LIN {X 0,Y 475.877,Z 329.982,A -85,B 0,C 180,E1 -7309.364,E2 -7309.364} C_VEL
LIN {X 0,Y 476.76,Z 310.728,A -85,B 0,C 180,E1 -7312.766,E2 -7312.766} C_VEL
LIN {X 0,Y 476.384,Z 304.918,A -85,B 0,C 180,E1 -7313.84,E2 -7313.84} C_VEL
LIN {X 0,Y 474.637,Z 296.366,A -85,B 0,C 180,E1 -7315.548,E2 -7315.548} C_VEL
LIN {X 0,Y 474.643,Z 296.366,A -85,B 0,C 180,E1 -7318.283,E2 -7318.283} C_VEL
LIN {X 0,Y 474.601,Z 296.37,A -85,B 0,C 180,E1 -7321.218,E2 -7321.218} C_VEL
LIN {X 0,Y 474.634,Z 296.366,A -85,B 0,C 180,E1 -7324.241,E2 -7324.241} C_VEL
LIN {X 0,Y 474.587,Z 296.366,A -85,B 0,C 180,E1 -7327.384,E2 -7327.384} C_VEL
LIN {X 0,Y 474.616,Z 296.363,A -85,B 0,C 180,E1 -7330.658,E2 -7330.658} C_VEL
LIN {X 0,Y 474.592,Z 296.363,A -85,B 0,C 180,E1 -7333.48,E2 -7333.48} C_VEL
LIN {X 0,Y 474.593,Z 296.37,A -85,B 0,C 180,E1 -7336.52,E2 -7336.52} C_VEL
LIN {X 0,Y 474.616,Z 296.36,A -85,B 0,C 180,E1 -7339.342,E2 -7339.342} C_VEL
LIN {X 0,Y 474.586,Z 296.37,A -85,B 0,C 180,E1 -7342.616,E2 -7342.616} C_VEL
LIN {X 0,Y 474.632,Z 296.357,A -85,B 0,C 180,E1 -7345.759,E2 -7345.759} C_VEL
LIN {X 0,Y 474.599,Z 296.366,A -85,B 0,C 180,E1 -7348.782,E2 -7348.782} C_VEL
LIN {X 0,Y 474.621,Z 296.358,A -85,B 0,C 180,E1 -7351.716,E2 -7351.716} C_VEL
LIN {X 0,Y 474.629,Z 296.36,A -85,B 0,C 180,E1 -7354.589,E2 -7354.589} C_VEL
LIN {X 0,Y 474.601,Z 296.368,A -85,B 0,C 180,E1 -7357.355,E2 -7357.355} C_VEL
LIN {X 0,Y 474.655,Z 296.355,A -85,B 0,C 180,E1 -7360.09,E2 -7360.09} C_VEL
LIN {X 0,Y 474.639,Z 296.356,A -85,B 0,C 180,E1 -7362.774,E2 -7362.774} C_VEL
LIN {X 0,Y 474.647,Z 296.362,A -85,B 0,C 180,E1 -7365.421,E2 -7365.421} C_VEL
LIN {X 0,Y 474.705,Z 296.35,A -85,B 0,C 180,E1 -7368.038,E2 -7368.038} C_VEL
LIN {X 0,Y 474.711,Z 296.35,A -85,B 0,C 180,E1 -7371.486,E2 -7371.486} C_VEL
LIN {X 0,Y 474.768,Z 296.344,A -85,B 0,C 180,E1 -7374.052,E2 -7374.052} C_VEL
LIN {X 0,Y 474.884,Z 296.325,A -85,B 0,C 180,E1 -7377.455,E2 -7377.455} C_VEL
LIN {X 0,Y 474.911,Z 296.327,A -85,B 0,C 180,E1 -7380,E2 -7380} C_VEL
LIN {X 0,Y 474.885,Z 296.329,A -85,B 0,C 180,E1 -7382.545,E2 -7382.545} C_VEL
LIN {X 0,Y 474.759,Z 296.342,A -85,B 0,C 180,E1 -7385.948,E2 -7385.948} C_VEL
LIN {X 0,Y 474.713,Z 296.351,A -85,B 0,C 180,E1 -7388.514,E2 -7388.514} C_VEL
LIN {X 0,Y 474.706,Z 296.35,A -85,B 0,C 180,E1 -7391.963,E2 -7391.963} C_VEL
LIN {X 0,Y 474.701,Z 296.35,A -85,B 0,C 180,E1 -7395.456,E2 -7395.456} C_VEL
LIN {X 0,Y 474.664,Z 296.36,A -85,B 0,C 180,E1 -7399.011,E2 -7399.011} C_VEL
LIN {X 0,Y 474.59,Z 296.361,A -85,B 0,C 180,E1 -7401.729,E2 -7401.729} C_VEL
LIN {X 0,Y 474.638,Z 296.358,A -85,B 0,C 180,E1 -7404.494,E2 -7404.494} C_VEL
LIN {X 0,Y 474.639,Z 296.361,A -85,B 0,C 180,E1 -7407.324,E2 -7407.324} C_VEL
LIN {X 0,Y 474.604,Z 296.361,A -85,B 0,C 180,E1 -7410.231,E2 -7410.231} C_VEL
LIN {X 0,Y 474.627,Z 296.365,A -85,B 0,C 180,E1 -7413.222,E2 -7413.222} C_VEL
LIN {X 0,Y 474.587,Z 296.364,A -85,B 0,C 180,E1 -7416.324,E2 -7416.324} C_VEL
LIN {X 0,Y 474.629,Z 296.365,A -85,B 0,C 180,E1 -7419.548,E2 -7419.548} C_VEL
LIN {X 0,Y 474.603,Z 296.364,A -85,B 0,C 180,E1 -7422.234,E2 -7422.234} C_VEL
LIN {X 0,Y 474.619,Z 296.363,A -85,B 0,C 180,E1 -7425.298,E2 -7425.298} C_VEL
LIN {X 0,Y 474.607,Z 296.368,A -85,B 0,C 180,E1 -7428.213,E2 -7428.213} C_VEL
LIN {X 0,Y 474.611,Z 296.367,A -85,B 0,C 180,E1 -7431.542,E2 -7431.542} C_VEL
LIN {X 0,Y 474.622,Z 296.365,A -85,B 0,C 180,E1 -7434.725,E2 -7434.725} C_VEL
LIN {X 0,Y 474.664,Z 296.454,A -85,B 0,C 180,E1 -7437.643,E2 -7437.643} C_VEL
LIN {X 0,Y 475.735,Z 302.876,A -85,B 0,C 180,E1 -7438.963,E2 -7438.963} C_VEL
LIN {X 0,Y 475.519,Z 316.144,A -85,B 0,C 180,E1 -7441.533,E2 -7441.533} C_VEL
LIN {X 0,Y 475.428,Z 319.942,A -85,B 0,C 180,E1 -7442.241,E2 -7442.241} C_VEL
LIN {X 0,Y 478.338,Z 335.26,A -85,B 0,C 180,E1 -7442.595,E2 -7442.595} C_VEL
LIN {X 0,Y 477.897,Z 378.829,A -85,B 0,C 180,E1 -7443.253,E2 -7443.253} C_VEL
LIN {X 0,Y 477.216,Z 384.671,A -85,B 0,C 180,E1 -7443.318,E2 -7443.318} C_VEL
LIN {X 0,Y 471.64,Z 403.685,A -85,B 0,C 180,E1 -7443.406,E2 -7443.406} C_VEL
LIN {X 0,Y 470.928,Z 409.529,A -85,B 0,C 180,E1 -7443.471,E2 -7443.471} C_VEL
LIN {X 0,Y 470.678,Z 429.482,A -85,B 0,C 180,E1 -7443.814,E2 -7443.814} C_VEL
LIN {X 0,Y 470.338,Z 442.898,A -85,B 0,C 180,E1 -7444.225,E2 -7444.225} C_VEL
LIN {X 0,Y 469.966,Z 454.955,A -85,B 0,C 180,E1 -7444.773,E2 -7444.773} C_VEL
LIN {X 0,Y 469.553,Z 466.283,A -85,B 0,C 180,E1 -7445.459,E2 -7445.459} C_VEL
LIN {X 0,Y 469.015,Z 478.056,A -85,B 0,C 180,E1 -7446.369,E2 -7446.369} C_VEL
LIN {X 0,Y 468.434,Z 488.504,A -85,B 0,C 180,E1 -7447.39,E2 -7447.39} C_VEL
LIN {X 0,Y 467.969,Z 498.494,A -85,B 0,C 180,E1 -7448.611,E2 -7448.611} C_VEL
LIN {X 0,Y 467.554,Z 506.223,A -85,B 0,C 180,E1 -7449.774,E2 -7449.774} C_VEL
LIN {X 0,Y 467.232,Z 513.348,A -85,B 0,C 180,E1 -7451.096,E2 -7451.096} C_VEL
LIN {X 0,Y 466.966,Z 519.248,A -85,B 0,C 180,E1 -7452.481,E2 -7452.481} C_VEL
LIN {X 0,Y 466.822,Z 523.709,A -85,B 0,C 180,E1 -7453.828,E2 -7453.828} C_VEL
LIN {X 0,Y 466.693,Z 527.025,A -85,B 0,C 180,E1 -7455.166,E2 -7455.166} C_VEL
LIN {X 0,Y 466.599,Z 528.656,A -85,B 0,C 180,E1 -7456.054,E2 -7456.054} C_VEL
LIN {X 0,Y 466.586,Z 529.862,A -85,B 0,C 180,E1 -7456.941,E2 -7456.941} C_VEL
LIN {X 0,Y 466.654,Z 530.818,A -85,B 0,C 180,E1 -7458.219,E2 -7458.219} C_VEL
LIN {X 0,Y 466.597,Z 530.896,A -85,B 0,C 180,E1 -7459.586,E2 -7459.586} C_VEL
LIN {X 0,Y 466.539,Z 530.442,A -85,B 0,C 180,E1 -7460.461,E2 -7460.461} C_VEL
LIN {X 0,Y 466.604,Z 529.545,A -85,B 0,C 180,E1 -7461.337,E2 -7461.337} C_VEL
LIN {X 0,Y 466.652,Z 528.255,A -85,B 0,C 180,E1 -7462.209,E2 -7462.209} C_VEL
LIN {X 0,Y 466.769,Z 525.339,A -85,B 0,C 180,E1 -7463.591,E2 -7463.591} C_VEL
LIN {X 0,Y 466.848,Z 521.789,A -85,B 0,C 180,E1 -7464.817,E2 -7464.817} C_VEL
LIN {X 0,Y 467.051,Z 516.937,A -85,B 0,C 180,E1 -7466.117,E2 -7466.117} C_VEL
LIN {X 0,Y 467.208,Z 510.853,A -85,B 0,C 180,E1 -7467.413,E2 -7467.413} C_VEL
LIN {X 0,Y 467.658,Z 503.274,A -85,B 0,C 180,E1 -7468.708,E2 -7468.708} C_VEL
LIN {X 0,Y 468.057,Z 493.792,A -85,B 0,C 180,E1 -7469.999,E2 -7469.999} C_VEL
LIN {X 0,Y 468.476,Z 484.032,A -85,B 0,C 180,E1 -7471.074,E2 -7471.074} C_VEL
LIN {X 0,Y 469.078,Z 473.058,A -85,B 0,C 180,E1 -7472.039,E2 -7472.039} C_VEL
LIN {X 0,Y 469.529,Z 462.354,A -85,B 0,C 180,E1 -7472.788,E2 -7472.788} C_VEL
LIN {X 0,Y 469.924,Z 449.501,A -85,B 0,C 180,E1 -7473.483,E2 -7473.483} C_VEL
LIN {X 0,Y 470.231,Z 437.091,A -85,B 0,C 180,E1 -7473.963,E2 -7473.963} C_VEL
LIN {X 0,Y 470.484,Z 424.139,A -85,B 0,C 180,E1 -7474.283,E2 -7474.283} C_VEL
LIN {X 0,Y 471.164,Z 335.118,A -85,B 0,C 180,E1 -7475.65,E2 -7475.65} C_VEL
LIN {X 0,Y 468.27,Z 320.023,A -85,B 0,C 180,E1 -7475.996,E2 -7475.996} C_VEL
LIN {X 0,Y 468.872,Z 306.744,A -85,B 0,C 180,E1 -7478.62,E2 -7478.62} C_VEL
LIN {X 0,Y 468.41,Z 301.4,A -85,B 0,C 180,E1 -7479.717,E2 -7479.717} C_VEL
LIN {X 0,Y 467.644,Z 297.234,A -85,B 0,C 180,E1 -7480.608,E2 -7480.608} C_VEL
LIN {X 0,Y 467.588,Z 297.24,A -85,B 0,C 180,E1 -7483.029,E2 -7483.029} C_VEL
LIN {X 0,Y 467.602,Z 297.24,A -85,B 0,C 180,E1 -7485.863,E2 -7485.863} C_VEL
LIN {X 0,Y 467.62,Z 297.231,A -85,B 0,C 180,E1 -7489.307,E2 -7489.307} C_VEL
LIN {X 0,Y 467.535,Z 297.249,A -85,B 0,C 180,E1 -7492.073,E2 -7492.073} C_VEL
LIN {X 0,Y 467.555,Z 297.24,A -85,B 0,C 180,E1 -7494.889,E2 -7494.889} C_VEL
LIN {X 0,Y 467.543,Z 297.242,A -85,B 0,C 180,E1 -7497.773,E2 -7497.773} C_VEL
LIN {X 0,Y 467.542,Z 297.242,A -85,B 0,C 180,E1 -7501.038,E2 -7501.038} C_VEL
LIN {X 0,Y 467.574,Z 297.241,A -85,B 0,C 180,E1 -7504.239,E2 -7504.239} C_VEL
LIN {X 0,Y 467.519,Z 297.245,A -85,B 0,C 180,E1 -7507.181,E2 -7507.181} C_VEL
LIN {X 0,Y 467.552,Z 297.242,A -85,B 0,C 180,E1 -7510.266,E2 -7510.266} C_VEL
LIN {X 0,Y 467.513,Z 297.249,A -85,B 0,C 180,E1 -7512.567,E2 -7512.567} C_VEL
LIN {X 0,Y 467.557,Z 297.245,A -85,B 0,C 180,E1 -7515.051,E2 -7515.051} C_VEL
LIN {X 0,Y 467.555,Z 297.244,A -85,B 0,C 180,E1 -7518.725,E2 -7518.725} C_VEL
LIN {X 0,Y 467.538,Z 297.241,A -85,B 0,C 180,E1 -7521.952,E2 -7521.952} C_VEL
LIN {X 0,Y 467.54,Z 297.249,A -85,B 0,C 180,E1 -7525.165,E2 -7525.165} C_VEL
LIN {X 0,Y 467.535,Z 297.241,A -85,B 0,C 180,E1 -7528.256,E2 -7528.256} C_VEL
LIN {X 0,Y 467.518,Z 297.25,A -85,B 0,C 180,E1 -7531.246,E2 -7531.246} C_VEL
LIN {X 0,Y 467.553,Z 297.239,A -85,B 0,C 180,E1 -7534.405,E2 -7534.405} C_VEL
LIN {X 0,Y 467.563,Z 297.239,A -85,B 0,C 180,E1 -7536.995,E2 -7536.995} C_VEL
LIN {X 0,Y 467.608,Z 297.24,A -85,B 0,C 180,E1 -7539.776,E2 -7539.776} C_VEL
LIN {X 0,Y 467.546,Z 297.241,A -85,B 0,C 180,E1 -7542.504,E2 -7542.504} C_VEL
LIN {X 0,Y 467.55,Z 297.24,A -85,B 0,C 180,E1 -7545.194,E2 -7545.194} C_VEL
LIN {X 0,Y 467.638,Z 297.236,A -85,B 0,C 180,E1 -7547.854,E2 -7547.854} C_VEL
LIN {X 0,Y 467.623,Z 297.231,A -85,B 0,C 180,E1 -7551.356,E2 -7551.356} C_VEL
LIN {X 0,Y 467.69,Z 297.228,A -85,B 0,C 180,E1 -7553.962,E2 -7553.962} C_VEL
LIN {X 0,Y 467.811,Z 297.207,A -85,B 0,C 180,E1 -7557.417,E2 -7557.417} C_VEL
LIN {X 0,Y 467.837,Z 297.208,A -85,B 0,C 180,E1 -7560,E2 -7560} C_VEL
LIN {X 0,Y 467.808,Z 297.214,A -85,B 0,C 180,E1 -7562.583,E2 -7562.583} C_VEL
LIN {X 0,Y 467.712,Z 297.222,A -85,B 0,C 180,E1 -7566.038,E2 -7566.038} C_VEL
LIN {X 0,Y 467.65,Z 297.236,A -85,B 0,C 180,E1 -7568.643,E2 -7568.643} C_VEL
LIN {X 0,Y 467.646,Z 297.229,A -85,B 0,C 180,E1 -7572.146,E2 -7572.146} C_VEL
LIN {X 0,Y 467.64,Z 297.228,A -85,B 0,C 180,E1 -7575.885,E2 -7575.885} C_VEL
LIN {X 0,Y 467.612,Z 297.236,A -85,B 0,C 180,E1 -7579.308,E2 -7579.308} C_VEL
LIN {X 0,Y 467.524,Z 297.243,A -85,B 0,C 180,E1 -7582.074,E2 -7582.074} C_VEL
LIN {X 0,Y 467.56,Z 297.244,A -85,B 0,C 180,E1 -7584.89,E2 -7584.89} C_VEL
LIN {X 0,Y 467.607,Z 297.234,A -85,B 0,C 180,E1 -7587.77,E2 -7587.77} C_VEL
LIN {X 0,Y 467.56,Z 297.243,A -85,B 0,C 180,E1 -7591.045,E2 -7591.045} C_VEL
LIN {X 0,Y 467.58,Z 297.236,A -85,B 0,C 180,E1 -7594.243,E2 -7594.243} C_VEL
LIN {X 0,Y 467.536,Z 297.245,A -85,B 0,C 180,E1 -7597.186,E2 -7597.186} C_VEL
LIN {X 0,Y 467.564,Z 297.239,A -85,B 0,C 180,E1 -7600.266,E2 -7600.266} C_VEL
LIN {X 0,Y 467.543,Z 297.249,A -85,B 0,C 180,E1 -7603.746,E2 -7603.746} C_VEL
LIN {X 0,Y 467.543,Z 297.243,A -85,B 0,C 180,E1 -7606.256,E2 -7606.256} C_VEL
LIN {X 0,Y 467.566,Z 297.244,A -85,B 0,C 180,E1 -7609.735,E2 -7609.735} C_VEL
LIN {X 0,Y 467.539,Z 297.241,A -85,B 0,C 180,E1 -7612.815,E2 -7612.815} C_VEL
LIN {X 0,Y 467.583,Z 297.243,A -85,B 0,C 180,E1 -7616.213,E2 -7616.213} C_VEL
LIN {X 0,Y 467.566,Z 297.237,A -85,B 0,C 180,E1 -7619.267,E2 -7619.267} C_VEL
LIN {X 0,Y 467.626,Z 297.238,A -85,B 0,C 180,E1 -7622.464,E2 -7622.464} C_VEL
LIN {X 0,Y 467.622,Z 297.399,A -85,B 0,C 180,E1 -7624.54,E2 -7624.54} C_VEL
LIN {X 0,Y 469.651,Z 308.372,A -85,B 0,C 180,E1 -7626.638,E2 -7626.638} C_VEL
LIN {X 0,Y 469.107,Z 323.782,A -85,B 0,C 180,E1 -7629.387,E2 -7629.387} C_VEL
LIN {X 0,Y 468.388,Z 341.681,A -85,B 0,C 180,E1 -7632.538,E2 -7632.538} C_VEL
LIN {X 0,Y 468.304,Z 344.549,A -85,B 0,C 180,E1 -7633.04,E2 -7633.04} C_VEL
LIN {X 0,Y 471.128,Z 364.408,A -85,B 0,C 180,E1 -7633.449,E2 -7633.449} C_VEL
LIN {X 0,Y 470.492,Z 452.851,A -85,B 0,C 180,E1 -7634.82,E2 -7634.82} C_VEL
LIN {X 0,Y 470.056,Z 466.105,A -85,B 0,C 180,E1 -7635.193,E2 -7635.193} C_VEL
LIN {X 0,Y 469.682,Z 478.282,A -85,B 0,C 180,E1 -7635.707,E2 -7635.707} C_VEL
LIN {X 0,Y 469.259,Z 489.754,A -85,B 0,C 180,E1 -7636.357,E2 -7636.357} C_VEL
LIN {X 0,Y 468.679,Z 501.743,A -85,B 0,C 180,E1 -7637.241,E2 -7637.241} C_VEL
LIN {X 0,Y 468.234,Z 512.089,A -85,B 0,C 180,E1 -7638.2,E2 -7638.2} C_VEL
LIN {X 0,Y 467.767,Z 520.715,A -85,B 0,C 180,E1 -7639.176,E2 -7639.176} C_VEL
LIN {X 0,Y 467.451,Z 528.671,A -85,B 0,C 180,E1 -7640.263,E2 -7640.263} C_VEL
LIN {X 0,Y 467.11,Z 536.44,A -85,B 0,C 180,E1 -7641.565,E2 -7641.565} C_VEL
LIN {X 0,Y 466.858,Z 543.58,A -85,B 0,C 180,E1 -7643.084,E2 -7643.084} C_VEL
LIN {X 0,Y 466.761,Z 548.334,A -85,B 0,C 180,E1 -7644.384,E2 -7644.384} C_VEL
LIN {X 0,Y 466.646,Z 551.963,A -85,B 0,C 180,E1 -7645.682,E2 -7645.682} C_VEL
LIN {X 0,Y 466.689,Z 553.839,A -85,B 0,C 180,E1 -7646.547,E2 -7646.547} C_VEL
LIN {X 0,Y 466.661,Z 555.246,A -85,B 0,C 180,E1 -7647.411,E2 -7647.411} C_VEL
LIN {X 0,Y 466.618,Z 556.86,A -85,B 0,C 180,E1 -7649.138,E2 -7649.138} C_VEL
LIN {X 0,Y 466.599,Z 557.083,A -85,B 0,C 180,E1 -7650.001,E2 -7650.001} C_VEL
LIN {X 0,Y 466.618,Z 556.875,A -85,B 0,C 180,E1 -7650.864,E2 -7650.864} C_VEL
LIN {X 0,Y 466.662,Z 555.28,A -85,B 0,C 180,E1 -7652.59,E2 -7652.59} C_VEL
LIN {X 0,Y 466.689,Z 553.892,A -85,B 0,C 180,E1 -7653.454,E2 -7653.454} C_VEL
LIN {X 0,Y 466.689,Z 550.965,A -85,B 0,C 180,E1 -7654.752,E2 -7654.752} C_VEL
LIN {X 0,Y 466.753,Z 547.007,A -85,B 0,C 180,E1 -7656.051,E2 -7656.051} C_VEL
LIN {X 0,Y 466.964,Z 540.93,A -85,B 0,C 180,E1 -7657.568,E2 -7657.568} C_VEL
LIN {X 0,Y 467.223,Z 534.286,A -85,B 0,C 180,E1 -7658.87,E2 -7658.87} C_VEL
LIN {X 0,Y 467.578,Z 526.045,A -85,B 0,C 180,E1 -7660.173,E2 -7660.173} C_VEL
LIN {X 0,Y 468.059,Z 517.625,A -85,B 0,C 180,E1 -7661.257,E2 -7661.257} C_VEL
LIN {X 0,Y 468.546,Z 507.619,A -85,B 0,C 180,E1 -7662.307,E2 -7662.307} C_VEL
LIN {X 0,Y 469.035,Z 495.703,A -85,B 0,C 180,E1 -7663.309,E2 -7663.309} C_VEL
LIN {X 0,Y 469.604,Z 483.932,A -85,B 0,C 180,E1 -7664.076,E2 -7664.076} C_VEL
LIN {X 0,Y 470.089,Z 471.867,A -85,B 0,C 180,E1 -7664.669,E2 -7664.669} C_VEL
LIN {X 0,Y 470.532,Z 458.762,A -85,B 0,C 180,E1 -7665.125,E2 -7665.125} C_VEL
LIN {X 0,Y 470.725,Z 446.209,A -85,B 0,C 180,E1 -7665.396,E2 -7665.396} C_VEL
LIN {X 0,Y 471.266,Z 362.018,A -85,B 0,C 180,E1 -7666.698,E2 -7666.698} C_VEL
LIN {X 0,Y 468.353,Z 344.319,A -85,B 0,C 180,E1 -7667.11,E2 -7667.11} C_VEL
LIN {X 0,Y 469.052,Z 328.4,A -85,B 0,C 180,E1 -7669.93,E2 -7669.93} C_VEL
LIN {X 0,Y 469.863,Z 311.951,A -85,B 0,C 180,E1 -7672.886,E2 -7672.886} C_VEL
LIN {X 0,Y 469.576,Z 306.893,A -85,B 0,C 180,E1 -7673.835,E2 -7673.835} C_VEL
LIN {X 0,Y 467.607,Z 297.241,A -85,B 0,C 180,E1 -7675.759,E2 -7675.759} C_VEL
LIN {X 0,Y 467.576,Z 297.245,A -85,B 0,C 180,E1 -7678.75,E2 -7678.75} C_VEL
LIN {X 0,Y 467.585,Z 297.245,A -85,B 0,C 180,E1 -7681.74,E2 -7681.74} C_VEL
LIN {X 0,Y 467.565,Z 297.242,A -85,B 0,C 180,E1 -7684.833,E2 -7684.833} C_VEL
LIN {X 0,Y 467.564,Z 297.246,A -85,B 0,C 180,E1 -7688.045,E2 -7688.045} C_VEL
LIN {X 0,Y 467.575,Z 297.237,A -85,B 0,C 180,E1 -7691.403,E2 -7691.403} C_VEL
LIN {X 0,Y 467.567,Z 297.24,A -85,B 0,C 180,E1 -7695.053,E2 -7695.053} C_VEL
LIN {X 0,Y 467.575,Z 297.243,A -85,B 0,C 180,E1 -7698.597,E2 -7698.597} C_VEL
LIN {X 0,Y 467.563,Z 297.237,A -85,B 0,C 180,E1 -7701.955,E2 -7701.955} C_VEL
LIN {X 0,Y 467.564,Z 297.241,A -85,B 0,C 180,E1 -7705.167,E2 -7705.167} C_VEL
LIN {X 0,Y 467.583,Z 297.235,A -85,B 0,C 180,E1 -7708.26,E2 -7708.26} C_VEL
LIN {X 0,Y 467.557,Z 297.242,A -85,B 0,C 180,E1 -7711.249,E2 -7711.249} C_VEL
LIN {X 0,Y 467.583,Z 297.236,A -85,B 0,C 180,E1 -7714.158,E2 -7714.158} C_VEL
LIN {X 0,Y 467.576,Z 297.242,A -85,B 0,C 180,E1 -7716.996,E2 -7716.996} C_VEL
LIN {X 0,Y 467.623,Z 297.233,A -85,B 0,C 180,E1 -7719.777,E2 -7719.777} C_VEL
LIN {X 0,Y 467.599,Z 297.232,A -85,B 0,C 180,E1 -7722.506,E2 -7722.506} C_VEL
LIN {X 0,Y 467.606,Z 297.236,A -85,B 0,C 180,E1 -7725.197,E2 -7725.197} C_VEL
LIN {X 0,Y 467.657,Z 297.23,A -85,B 0,C 180,E1 -7727.855,E2 -7727.855} C_VEL
LIN {X 0,Y 467.669,Z 297.226,A -85,B 0,C 180,E1 -7731.357,E2 -7731.357} C_VEL
LIN {X 0,Y 467.732,Z 297.222,A -85,B 0,C 180,E1 -7733.963,E2 -7733.963} C_VEL
LIN {X 0,Y 467.848,Z 297.201,A -85,B 0,C 180,E1 -7737.417,E2 -7737.417} C_VEL
LIN {X 0,Y 467.881,Z 297.202,A -85,B 0,C 180,E1 -7740,E2 -7740} C_VEL
LIN {X 0,Y 467.851,Z 297.204,A -85,B 0,C 180,E1 -7742.583,E2 -7742.583} C_VEL
LIN {X 0,Y 467.721,Z 297.22,A -85,B 0,C 180,E1 -7746.038,E2 -7746.038} C_VEL
LIN {X 0,Y 467.671,Z 297.226,A -85,B 0,C 180,E1 -7748.643,E2 -7748.643} C_VEL
LIN {X 0,Y 467.657,Z 297.23,A -85,B 0,C 180,E1 -7752.146,E2 -7752.146} C_VEL
LIN {X 0,Y 467.64,Z 297.229,A -85,B 0,C 180,E1 -7755.695,E2 -7755.695} C_VEL
LIN {X 0,Y 467.624,Z 297.233,A -85,B 0,C 180,E1 -7759.308,E2 -7759.308} C_VEL
LIN {X 0,Y 467.536,Z 297.239,A -85,B 0,C 180,E1 -7762.074,E2 -7762.074} C_VEL
LIN {X 0,Y 467.585,Z 297.24,A -85,B 0,C 180,E1 -7764.889,E2 -7764.889} C_VEL
LIN {X 0,Y 467.582,Z 297.235,A -85,B 0,C 180,E1 -7767.772,E2 -7767.772} C_VEL
LIN {X 0,Y 467.57,Z 297.243,A -85,B 0,C 180,E1 -7771.045,E2 -7771.045} C_VEL
LIN {X 0,Y 467.579,Z 297.235,A -85,B 0,C 180,E1 -7774.24,E2 -7774.24} C_VEL
LIN {X 0,Y 467.546,Z 297.246,A -85,B 0,C 180,E1 -7777.186,E2 -7777.186} C_VEL
LIN {X 0,Y 467.573,Z 297.239,A -85,B 0,C 180,E1 -7780.266,E2 -7780.266} C_VEL
LIN {X 0,Y 467.552,Z 297.247,A -85,B 0,C 180,E1 -7783.745,E2 -7783.745} C_VEL
LIN {X 0,Y 467.549,Z 297.246,A -85,B 0,C 180,E1 -7786.255,E2 -7786.255} C_VEL
LIN {X 0,Y 467.562,Z 297.243,A -85,B 0,C 180,E1 -7789.734,E2 -7789.734} C_VEL
LIN {X 0,Y 467.544,Z 297.246,A -85,B 0,C 180,E1 -7792.815,E2 -7792.815} C_VEL
LIN {X 0,Y 467.58,Z 297.242,A -85,B 0,C 180,E1 -7795.76,E2 -7795.76} C_VEL
LIN {X 0,Y 467.623,Z 297.363,A -85,B 0,C 180,E1 -7797.433,E2 -7797.433} C_VEL
LIN {X 0,Y 468.78,Z 303.442,A -85,B 0,C 180,E1 -7798.711,E2 -7798.711} C_VEL
LIN {X 0,Y 468.609,Z 315.461,A -85,B 0,C 180,E1 -7801.074,E2 -7801.074} C_VEL
LIN {X 0,Y 468.493,Z 320.009,A -85,B 0,C 180,E1 -7801.958,E2 -7801.958} C_VEL
LIN {X 0,Y 471.597,Z 336.382,A -85,B 0,C 180,E1 -7802.345,E2 -7802.345} C_VEL
LIN {X 0,Y 470.928,Z 409.529,A -85,B 0,C 180,E1 -7803.471,E2 -7803.471} C_VEL
LIN {X 0,Y 470.178,Z 415.387,A -85,B 0,C 180,E1 -7803.533,E2 -7803.533} C_VEL
LIN {X 0,Y 464.787,Z 432.398,A -85,B 0,C 180,E1 -7803.665,E2 -7803.665} C_VEL
LIN {X 0,Y 463.746,Z 438.123,A -85,B 0,C 180,E1 -7803.802,E2 -7803.802} C_VEL
LIN {X 0,Y 463.658,Z 439.971,A -85,B 0,C 180,E1 -7803.867,E2 -7803.867} C_VEL
LIN {X 0,Y 463.211,Z 453.323,A -85,B 0,C 180,E1 -7804.439,E2 -7804.439} C_VEL
LIN {X 0,Y 462.822,Z 464.254,A -85,B 0,C 180,E1 -7805.077,E2 -7805.077} C_VEL
LIN {X 0,Y 462.26,Z 475.488,A -85,B 0,C 180,E1 -7805.917,E2 -7805.917} C_VEL
LIN {X 0,Y 461.687,Z 486.185,A -85,B 0,C 180,E1 -7806.922,E2 -7806.922} C_VEL
LIN {X 0,Y 461.159,Z 495.435,A -85,B 0,C 180,E1 -7807.993,E2 -7807.993} C_VEL
LIN {X 0,Y 460.702,Z 504.069,A -85,B 0,C 180,E1 -7809.226,E2 -7809.226} C_VEL
LIN {X 0,Y 460.295,Z 511.931,A -85,B 0,C 180,E1 -7810.627,E2 -7810.627} C_VEL
LIN {X 0,Y 459.962,Z 518.881,A -85,B 0,C 180,E1 -7812.206,E2 -7812.206} C_VEL
LIN {X 0,Y 459.755,Z 523.47,A -85,B 0,C 180,E1 -7813.572,E2 -7813.572} C_VEL
LIN {X 0,Y 459.633,Z 526.91,A -85,B 0,C 180,E1 -7814.933,E2 -7814.933} C_VEL
LIN {X 0,Y 459.531,Z 528.601,A -85,B 0,C 180,E1 -7815.835,E2 -7815.835} C_VEL
LIN {X 0,Y 459.5,Z 529.872,A -85,B 0,C 180,E1 -7816.736,E2 -7816.736} C_VEL
LIN {X 0,Y 459.567,Z 531.003,A -85,B 0,C 180,E1 -7818.164,E2 -7818.164} C_VEL
LIN {X 0,Y 459.5,Z 531.123,A -85,B 0,C 180,E1 -7819.424,E2 -7819.424} C_VEL
LIN {X 0,Y 459.446,Z 530.742,A -85,B 0,C 180,E1 -7820.313,E2 -7820.313} C_VEL
LIN {X 0,Y 459.499,Z 529.939,A -85,B 0,C 180,E1 -7821.202,E2 -7821.202} C_VEL
LIN {X 0,Y 459.545,Z 528.705,A -85,B 0,C 180,E1 -7822.088,E2 -7822.088} C_VEL
LIN {X 0,Y 459.677,Z 525.611,A -85,B 0,C 180,E1 -7823.614,E2 -7823.614} C_VEL
LIN {X 0,Y 459.786,Z 521.053,A -85,B 0,C 180,E1 -7825.177,E2 -7825.177} C_VEL
LIN {X 0,Y 460.035,Z 515.938,A -85,B 0,C 180,E1 -7826.496,E2 -7826.496} C_VEL
LIN {X 0,Y 460.233,Z 509.528,A -85,B 0,C 180,E1 -7827.812,E2 -7827.812} C_VEL
LIN {X 0,Y 460.745,Z 501.531,A -85,B 0,C 180,E1 -7829.125,E2 -7829.125} C_VEL
LIN {X 0,Y 461.057,Z 493.425,A -85,B 0,C 180,E1 -7830.218,E2 -7830.218} C_VEL
LIN {X 0,Y 461.588,Z 483.524,A -85,B 0,C 180,E1 -7831.308,E2 -7831.308} C_VEL
LIN {X 0,Y 462.112,Z 473.739,A -85,B 0,C 180,E1 -7832.178,E2 -7832.178} C_VEL
LIN {X 0,Y 462.641,Z 461.402,A -85,B 0,C 180,E1 -7833.047,E2 -7833.047} C_VEL
LIN {X 0,Y 463.034,Z 449.332,A -85,B 0,C 180,E1 -7833.698,E2 -7833.698} C_VEL
LIN {X 0,Y 463.346,Z 436.694,A -85,B 0,C 180,E1 -7834.185,E2 -7834.185} C_VEL
LIN {X 0,Y 463.641,Z 423.318,A -85,B 0,C 180,E1 -7834.509,E2 -7834.509} C_VEL
LIN {X 0,Y 464.294,Z 335.908,A -85,B 0,C 180,E1 -7835.87,E2 -7835.87} C_VEL
LIN {X 0,Y 461.273,Z 320.211,A -85,B 0,C 180,E1 -7836.231,E2 -7836.231} C_VEL
LIN {X 0,Y 461.915,Z 307.587,A -85,B 0,C 180,E1 -7838.751,E2 -7838.751} C_VEL
LIN {X 0,Y 461.362,Z 302.242,A -85,B 0,C 180,E1 -7839.867,E2 -7839.867} C_VEL
LIN {X 0,Y 460.595,Z 298.112,A -85,B 0,C 180,E1 -7840.772,E2 -7840.772} C_VEL
LIN {X 0,Y 460.543,Z 298.119,A -85,B 0,C 180,E1 -7843.232,E2 -7843.232} C_VEL
LIN {X 0,Y 460.559,Z 298.119,A -85,B 0,C 180,E1 -7845.977,E2 -7845.977} C_VEL
LIN {X 0,Y 460.567,Z 298.112,A -85,B 0,C 180,E1 -7849.615,E2 -7849.615} C_VEL
LIN {X 0,Y 460.511,Z 298.121,A -85,B 0,C 180,E1 -7852.428,E2 -7852.428} C_VEL
LIN {X 0,Y 460.532,Z 298.116,A -85,B 0,C 180,E1 -7855.791,E2 -7855.791} C_VEL
LIN {X 0,Y 460.515,Z 298.116,A -85,B 0,C 180,E1 -7859.232,E2 -7859.232} C_VEL
LIN {X 0,Y 460.516,Z 298.122,A -85,B 0,C 180,E1 -7862.284,E2 -7862.284} C_VEL
LIN {X 0,Y 460.502,Z 298.118,A -85,B 0,C 180,E1 -7865.445,E2 -7865.445} C_VEL
LIN {X 0,Y 460.494,Z 298.125,A -85,B 0,C 180,E1 -7868.889,E2 -7868.889} C_VEL
LIN {X 0,Y 460.498,Z 298.118,A -85,B 0,C 180,E1 -7871.597,E2 -7871.597} C_VEL
LIN {X 0,Y 460.505,Z 298.122,A -85,B 0,C 180,E1 -7874.589,E2 -7874.589} C_VEL
LIN {X 0,Y 460.468,Z 298.122,A -85,B 0,C 180,E1 -7877.812,E2 -7877.812} C_VEL
LIN {X 0,Y 460.504,Z 298.117,A -85,B 0,C 180,E1 -7880.134,E2 -7880.134} C_VEL
LIN {X 0,Y 460.454,Z 298.128,A -85,B 0,C 180,E1 -7883.468,E2 -7883.468} C_VEL
LIN {X 0,Y 460.493,Z 298.12,A -85,B 0,C 180,E1 -7886.672,E2 -7886.672} C_VEL
LIN {X 0,Y 460.471,Z 298.125,A -85,B 0,C 180,E1 -7889.757,E2 -7889.757} C_VEL
LIN {X 0,Y 460.476,Z 298.121,A -85,B 0,C 180,E1 -7892.75,E2 -7892.75} C_VEL
LIN {X 0,Y 460.504,Z 298.125,A -85,B 0,C 180,E1 -7895.665,E2 -7895.665} C_VEL
LIN {X 0,Y 460.513,Z 298.116,A -85,B 0,C 180,E1 -7898.578,E2 -7898.578} C_VEL
LIN {X 0,Y 460.53,Z 298.117,A -85,B 0,C 180,E1 -7901.308,E2 -7901.308} C_VEL
LIN {X 0,Y 460.511,Z 298.122,A -85,B 0,C 180,E1 -7904.055,E2 -7904.055} C_VEL
LIN {X 0,Y 460.594,Z 298.111,A -85,B 0,C 180,E1 -7907.665,E2 -7907.665} C_VEL
LIN {X 0,Y 460.578,Z 298.108,A -85,B 0,C 180,E1 -7911.223,E2 -7911.223} C_VEL
LIN {X 0,Y 460.656,Z 298.103,A -85,B 0,C 180,E1 -7913.869,E2 -7913.869} C_VEL
LIN {X 0,Y 460.755,Z 298.086,A -85,B 0,C 180,E1 -7917.377,E2 -7917.377} C_VEL
LIN {X 0,Y 460.806,Z 298.084,A -85,B 0,C 180,E1 -7920,E2 -7920} C_VEL
LIN {X 0,Y 460.752,Z 298.092,A -85,B 0,C 180,E1 -7922.623,E2 -7922.623} C_VEL
LIN {X 0,Y 460.678,Z 298.099,A -85,B 0,C 180,E1 -7926.13,E2 -7926.13} C_VEL
LIN {X 0,Y 460.601,Z 298.112,A -85,B 0,C 180,E1 -7928.777,E2 -7928.777} C_VEL
LIN {X 0,Y 460.587,Z 298.111,A -85,B 0,C 180,E1 -7932.435,E2 -7932.435} C_VEL
LIN {X 0,Y 460.592,Z 298.106,A -85,B 0,C 180,E1 -7935.998,E2 -7935.998} C_VEL
LIN {X 0,Y 460.558,Z 298.112,A -85,B 0,C 180,E1 -7939.616,E2 -7939.616} C_VEL
LIN {X 0,Y 460.501,Z 298.119,A -85,B 0,C 180,E1 -7942.429,E2 -7942.429} C_VEL
LIN {X 0,Y 460.537,Z 298.114,A -85,B 0,C 180,E1 -7945.796,E2 -7945.796} C_VEL
LIN {X 0,Y 460.541,Z 298.113,A -85,B 0,C 180,E1 -7948.234,E2 -7948.234} C_VEL
LIN {X 0,Y 460.513,Z 298.124,A -85,B 0,C 180,E1 -7951.283,E2 -7951.283} C_VEL
LIN {X 0,Y 460.523,Z 298.115,A -85,B 0,C 180,E1 -7954.506,E2 -7954.506} C_VEL
LIN {X 0,Y 460.492,Z 298.126,A -85,B 0,C 180,E1 -7957.624,E2 -7957.624} C_VEL
LIN {X 0,Y 460.521,Z 298.116,A -85,B 0,C 180,E1 -7961.012,E2 -7961.012} C_VEL
LIN {X 0,Y 460.506,Z 298.117,A -85,B 0,C 180,E1 -7964.59,E2 -7964.59} C_VEL
LIN {X 0,Y 460.499,Z 298.126,A -85,B 0,C 180,E1 -7967.817,E2 -7967.817} C_VEL
LIN {X 0,Y 460.527,Z 298.115,A -85,B 0,C 180,E1 -7971.105,E2 -7971.105} C_VEL
LIN {X 0,Y 460.505,Z 298.12,A -85,B 0,C 180,E1 -7974.555,E2 -7974.555} C_VEL
LIN {X 0,Y 460.528,Z 298.117,A -85,B 0,C 180,E1 -7977.717,E2 -7977.717} C_VEL
LIN {X 0,Y 460.536,Z 298.116,A -85,B 0,C 180,E1 -7980.77,E2 -7980.77} C_VEL
LIN {X 0,Y 460.54,Z 298.117,A -85,B 0,C 180,E1 -7983.734,E2 -7983.734} C_VEL
LIN {X 0,Y 460.557,Z 298.171,A -85,B 0,C 180,E1 -7984.342,E2 -7984.342} C_VEL
LIN {X 0,Y 462.636,Z 309.333,A -85,B 0,C 180,E1 -7986.508,E2 -7986.508} C_VEL
LIN {X 0,Y 462.332,Z 319.188,A -85,B 0,C 180,E1 -7988.298,E2 -7988.298} C_VEL
LIN {X 0,Y 461.585,Z 337.508,A -85,B 0,C 180,E1 -7991.584,E2 -7991.584} C_VEL
LIN {X 0,Y 461.292,Z 344.371,A -85,B 0,C 180,E1 -7992.803,E2 -7992.803} C_VEL
LIN {X 0,Y 464.259,Z 364.445,A -85,B 0,C 180,E1 -7993.223,E2 -7993.223} C_VEL
LIN {X 0,Y 463.607,Z 452.914,A -85,B 0,C 180,E1 -7994.617,E2 -7994.617} C_VEL
LIN {X 0,Y 463.142,Z 466.852,A -85,B 0,C 180,E1 -7995.023,E2 -7995.023} C_VEL
LIN {X 0,Y 462.704,Z 479.848,A -85,B 0,C 180,E1 -7995.599,E2 -7995.599} C_VEL
LIN {X 0,Y 462.188,Z 492.458,A -85,B 0,C 180,E1 -7996.368,E2 -7996.368} C_VEL
LIN {X 0,Y 461.61,Z 503.666,A -85,B 0,C 180,E1 -7997.245,E2 -7997.245} C_VEL
LIN {X 0,Y 461.204,Z 512.777,A -85,B 0,C 180,E1 -7998.129,E2 -7998.129} C_VEL
LIN {X 0,Y 460.669,Z 522.089,A -85,B 0,C 180,E1 -7999.23,E2 -7999.23} C_VEL
LIN {X 0,Y 460.278,Z 531.127,A -85,B 0,C 180,E1 -8000.553,E2 -8000.553} C_VEL
LIN {X 0,Y 459.951,Z 538.401,A -85,B 0,C 180,E1 -8001.875,E2 -8001.875} C_VEL
LIN {X 0,Y 459.744,Z 544.502,A -85,B 0,C 180,E1 -8003.273,E2 -8003.273} C_VEL
LIN {X 0,Y 459.65,Z 549.414,A -85,B 0,C 180,E1 -8004.737,E2 -8004.737} C_VEL
LIN {X 0,Y 459.564,Z 551.727,A -85,B 0,C 180,E1 -8005.615,E2 -8005.615} C_VEL
LIN {X 0,Y 459.584,Z 553.611,A -85,B 0,C 180,E1 -8006.494,E2 -8006.494} C_VEL
LIN {X 0,Y 459.583,Z 555.029,A -85,B 0,C 180,E1 -8007.371,E2 -8007.371} C_VEL
LIN {X 0,Y 459.521,Z 556.653,A -85,B 0,C 180,E1 -8009.124,E2 -8009.124} C_VEL
LIN {X 0,Y 459.53,Z 556.884,A -85,B 0,C 180,E1 -8010.001,E2 -8010.001} C_VEL
LIN {X 0,Y 459.521,Z 556.684,A -85,B 0,C 180,E1 -8010.877,E2 -8010.877} C_VEL
LIN {X 0,Y 459.584,Z 555.101,A -85,B 0,C 180,E1 -8012.63,E2 -8012.63} C_VEL
LIN {X 0,Y 459.583,Z 553.719,A -85,B 0,C 180,E1 -8013.507,E2 -8013.507} C_VEL
LIN {X 0,Y 459.617,Z 550.804,A -85,B 0,C 180,E1 -8014.825,E2 -8014.825} C_VEL
LIN {X 0,Y 459.713,Z 545.851,A -85,B 0,C 180,E1 -8016.43,E2 -8016.43} C_VEL
LIN {X 0,Y 459.924,Z 539.797,A -85,B 0,C 180,E1 -8017.905,E2 -8017.905} C_VEL
LIN {X 0,Y 460.225,Z 532.95,A -85,B 0,C 180,E1 -8019.227,E2 -8019.227} C_VEL
LIN {X 0,Y 460.618,Z 524.418,A -85,B 0,C 180,E1 -8020.551,E2 -8020.551} C_VEL
LIN {X 0,Y 461.185,Z 515.667,A -85,B 0,C 180,E1 -8021.65,E2 -8021.65} C_VEL
LIN {X 0,Y 461.746,Z 505.954,A -85,B 0,C 180,E1 -8022.651,E2 -8022.651} C_VEL
LIN {X 0,Y 462.135,Z 495.627,A -85,B 0,C 180,E1 -8023.522,E2 -8023.522} C_VEL
LIN {X 0,Y 462.738,Z 484.115,A -85,B 0,C 180,E1 -8024.289,E2 -8024.289} C_VEL
LIN {X 0,Y 463.248,Z 472.184,A -85,B 0,C 180,E1 -8024.89,E2 -8024.89} C_VEL
LIN {X 0,Y 463.718,Z 459.3,A -85,B 0,C 180,E1 -8025.353,E2 -8025.353} C_VEL
LIN {X 0,Y 463.945,Z 445.692,A -85,B 0,C 180,E1 -8025.655,E2 -8025.655} C_VEL
LIN {X 0,Y 464.523,Z 362.908,A -85,B 0,C 180,E1 -8026.955,E2 -8026.955} C_VEL
LIN {X 0,Y 461.43,Z 344.092,A -85,B 0,C 180,E1 -8027.406,E2 -8027.406} C_VEL
LIN {X 0,Y 462.147,Z 328.355,A -85,B 0,C 180,E1 -8030.241,E2 -8030.241} C_VEL
LIN {X 0,Y 462.959,Z 311.927,A -85,B 0,C 180,E1 -8033.247,E2 -8033.247} C_VEL
LIN {X 0,Y 462.334,Z 306.874,A -85,B 0,C 180,E1 -8034.232,E2 -8034.232} C_VEL
LIN {X 0,Y 460.543,Z 298.121,A -85,B 0,C 180,E1 -8036.024,E2 -8036.024} C_VEL
LIN {X 0,Y 460.552,Z 298.122,A -85,B 0,C 180,E1 -8038.233,E2 -8038.233} C_VEL
LIN {X 0,Y 460.523,Z 298.125,A -85,B 0,C 180,E1 -8041.283,E2 -8041.283} C_VEL
LIN {X 0,Y 460.533,Z 298.12,A -85,B 0,C 180,E1 -8044.505,E2 -8044.505} C_VEL
LIN {X 0,Y 460.5,Z 298.123,A -85,B 0,C 180,E1 -8047.624,E2 -8047.624} C_VEL
LIN {X 0,Y 460.529,Z 298.115,A -85,B 0,C 180,E1 -8051.012,E2 -8051.012} C_VEL
LIN {X 0,Y 460.513,Z 298.123,A -85,B 0,C 180,E1 -8054.589,E2 -8054.589} C_VEL
LIN {X 0,Y 460.505,Z 298.12,A -85,B 0,C 180,E1 -8057.817,E2 -8057.817} C_VEL
LIN {X 0,Y 460.521,Z 298.119,A -85,B 0,C 180,E1 -8060.136,E2 -8060.136} C_VEL
LIN {X 0,Y 460.474,Z 298.122,A -85,B 0,C 180,E1 -8063.47,E2 -8063.47} C_VEL
LIN {X 0,Y 460.528,Z 298.121,A -85,B 0,C 180,E1 -8066.675,E2 -8066.675} C_VEL
LIN {X 0,Y 460.508,Z 298.118,A -85,B 0,C 180,E1 -8069.76,E2 -8069.76} C_VEL
LIN {X 0,Y 460.535,Z 298.117,A -85,B 0,C 180,E1 -8072.754,E2 -8072.754} C_VEL
LIN {X 0,Y 460.522,Z 298.117,A -85,B 0,C 180,E1 -8075.667,E2 -8075.667} C_VEL
LIN {X 0,Y 460.522,Z 298.115,A -85,B 0,C 180,E1 -8078.578,E2 -8078.578} C_VEL
LIN {X 0,Y 460.587,Z 298.115,A -85,B 0,C 180,E1 -8081.311,E2 -8081.311} C_VEL
LIN {X 0,Y 460.605,Z 298.105,A -85,B 0,C 180,E1 -8084.059,E2 -8084.059} C_VEL
LIN {X 0,Y 460.61,Z 298.107,A -85,B 0,C 180,E1 -8087.666,E2 -8087.666} C_VEL
LIN {X 0,Y 460.619,Z 298.103,A -85,B 0,C 180,E1 -8091.224,E2 -8091.224} C_VEL
LIN {X 0,Y 460.698,Z 298.1,A -85,B 0,C 180,E1 -8093.87,E2 -8093.87} C_VEL
LIN {X 0,Y 460.789,Z 298.08,A -85,B 0,C 180,E1 -8097.378,E2 -8097.378} C_VEL
LIN {X 0,Y 460.851,Z 298.077,A -85,B 0,C 180,E1 -8100,E2 -8100} C_VEL
LIN {X 0,Y 460.791,Z 298.083,A -85,B 0,C 180,E1 -8102.623,E2 -8102.623} C_VEL
LIN {X 0,Y 460.686,Z 298.097,A -85,B 0,C 180,E1 -8106.13,E2 -8106.13} C_VEL
LIN {X 0,Y 460.621,Z 298.103,A -85,B 0,C 180,E1 -8108.777,E2 -8108.777} C_VEL
LIN {X 0,Y 460.615,Z 298.111,A -85,B 0,C 180,E1 -8112.445,E2 -8112.445} C_VEL
LIN {X 0,Y 460.602,Z 298.107,A -85,B 0,C 180,E1 -8115.998,E2 -8115.998} C_VEL
LIN {X 0,Y 460.57,Z 298.11,A -85,B 0,C 180,E1 -8119.616,E2 -8119.616} C_VEL
LIN {X 0,Y 460.512,Z 298.116,A -85,B 0,C 180,E1 -8122.429,E2 -8122.429} C_VEL
LIN {X 0,Y 460.55,Z 298.111,A -85,B 0,C 180,E1 -8125.797,E2 -8125.797} C_VEL
LIN {X 0,Y 460.529,Z 298.112,A -85,B 0,C 180,E1 -8128.235,E2 -8128.235} C_VEL
LIN {X 0,Y 460.522,Z 298.12,A -85,B 0,C 180,E1 -8131.283,E2 -8131.283} C_VEL
LIN {X 0,Y 460.525,Z 298.114,A -85,B 0,C 180,E1 -8134.504,E2 -8134.504} C_VEL
LIN {X 0,Y 460.502,Z 298.125,A -85,B 0,C 180,E1 -8137.624,E2 -8137.624} C_VEL
LIN {X 0,Y 460.538,Z 298.116,A -85,B 0,C 180,E1 -8140.268,E2 -8140.268} C_VEL
LIN {X 0,Y 460.512,Z 298.122,A -85,B 0,C 180,E1 -8143.375,E2 -8143.375} C_VEL
LIN {X 0,Y 460.506,Z 298.121,A -85,B 0,C 180,E1 -8146.625,E2 -8146.625} C_VEL
LIN {X 0,Y 460.528,Z 298.119,A -85,B 0,C 180,E1 -8149.733,E2 -8149.733} C_VEL
LIN {X 0,Y 460.499,Z 298.124,A -85,B 0,C 180,E1 -8152.525,E2 -8152.525} C_VEL
LIN {X 0,Y 460.539,Z 298.119,A -85,B 0,C 180,E1 -8155.623,E2 -8155.623} C_VEL
LIN {X 0,Y 460.564,Z 298.29,A -85,B 0,C 180,E1 -8157.214,E2 -8157.214} C_VEL
LIN {X 0,Y 461.921,Z 305.985,A -85,B 0,C 180,E1 -8158.848,E2 -8158.848} C_VEL
LIN {X 0,Y 461.609,Z 319.843,A -85,B 0,C 180,E1 -8161.598,E2 -8161.598} C_VEL
LIN {X 0,Y 461.585,Z 320.143,A -85,B 0,C 180,E1 -8161.656,E2 -8161.656} C_VEL
LIN {X 0,Y 464.807,Z 336.126,A -85,B 0,C 180,E1 -8162.061,E2 -8162.061} C_VEL
LIN {X 0,Y 463.949,Z 428.274,A -85,B 0,C 180,E1 -8163.529,E2 -8163.529} C_VEL
LIN {X 0,Y 463.658,Z 439.971,A -85,B 0,C 180,E1 -8163.867,E2 -8163.867} C_VEL
LIN {X 0,Y 462.935,Z 443.78,A -85,B 0,C 180,E1 -8163.983,E2 -8163.983} C_VEL
LIN {X 0,Y 459.977,Z 449.761,A -85,B 0,C 180,E1 -8164.134,E2 -8164.134} C_VEL
LIN {X 0,Y 456.955,Z 455.622,A -85,B 0,C 180,E1 -8164.322,E2 -8164.322} C_VEL
LIN {X 0,Y 456.161,Z 459.237,A -85,B 0,C 180,E1 -8164.506,E2 -8164.506} C_VEL
LIN {X 0,Y 455.66,Z 470.474,A -85,B 0,C 180,E1 -8165.268,E2 -8165.268} C_VEL
LIN {X 0,Y 455.054,Z 481.577,A -85,B 0,C 180,E1 -8166.223,E2 -8166.223} C_VEL
LIN {X 0,Y 454.463,Z 491.273,A -85,B 0,C 180,E1 -8167.256,E2 -8167.256} C_VEL
LIN {X 0,Y 453.944,Z 500.802,A -85,B 0,C 180,E1 -8168.516,E2 -8168.516} C_VEL
LIN {X 0,Y 453.452,Z 508.784,A -85,B 0,C 180,E1 -8169.827,E2 -8169.827} C_VEL
LIN {X 0,Y 453.106,Z 515.129,A -85,B 0,C 180,E1 -8171.114,E2 -8171.114} C_VEL
LIN {X 0,Y 452.864,Z 520.184,A -85,B 0,C 180,E1 -8172.384,E2 -8172.384} C_VEL
LIN {X 0,Y 452.659,Z 524.516,A -85,B 0,C 180,E1 -8173.771,E2 -8173.771} C_VEL
LIN {X 0,Y 452.589,Z 526.792,A -85,B 0,C 180,E1 -8174.693,E2 -8174.693} C_VEL
LIN {X 0,Y 452.479,Z 528.552,A -85,B 0,C 180,E1 -8175.61,E2 -8175.61} C_VEL
LIN {X 0,Y 452.413,Z 529.879,A -85,B 0,C 180,E1 -8176.525,E2 -8176.525} C_VEL
LIN {X 0,Y 452.478,Z 531.19,A -85,B 0,C 180,E1 -8178.108,E2 -8178.108} C_VEL
LIN {X 0,Y 452.406,Z 531.35,A -85,B 0,C 180,E1 -8179.256,E2 -8179.256} C_VEL
LIN {X 0,Y 452.408,Z 530.302,A -85,B 0,C 180,E1 -8181.063,E2 -8181.063} C_VEL
LIN {X 0,Y 452.457,Z 529.149,A -85,B 0,C 180,E1 -8181.963,E2 -8181.963} C_VEL
LIN {X 0,Y 452.605,Z 525.927,A -85,B 0,C 180,E1 -8183.613,E2 -8183.613} C_VEL
LIN {X 0,Y 452.7,Z 521.729,A -85,B 0,C 180,E1 -8185.101,E2 -8185.101} C_VEL
LIN {X 0,Y 452.946,Z 516.751,A -85,B 0,C 180,E1 -8186.441,E2 -8186.441} C_VEL
LIN {X 0,Y 453.165,Z 510.522,A -85,B 0,C 180,E1 -8187.777,E2 -8187.777} C_VEL
LIN {X 0,Y 453.666,Z 502.709,A -85,B 0,C 180,E1 -8189.112,E2 -8189.112} C_VEL
LIN {X 0,Y 454.01,Z 494.79,A -85,B 0,C 180,E1 -8190.221,E2 -8190.221} C_VEL
LIN {X 0,Y 454.464,Z 485.141,A -85,B 0,C 180,E1 -8191.329,E2 -8191.329} C_VEL
LIN {X 0,Y 455.147,Z 474.368,A -85,B 0,C 180,E1 -8192.322,E2 -8192.322} C_VEL
LIN {X 0,Y 455.698,Z 462.143,A -85,B 0,C 180,E1 -8193.204,E2 -8193.204} C_VEL
LIN {X 0,Y 456.1,Z 450.221,A -85,B 0,C 180,E1 -8193.865,E2 -8193.865} C_VEL
LIN {X 0,Y 456.428,Z 437.993,A -85,B 0,C 180,E1 -8194.36,E2 -8194.36} C_VEL
LIN {X 0,Y 456.713,Z 425.357,A -85,B 0,C 180,E1 -8194.688,E2 -8194.688} C_VEL
LIN {X 0,Y 457.448,Z 336.537,A -85,B 0,C 180,E1 -8196.095,E2 -8196.095} C_VEL
LIN {X 0,Y 454.342,Z 320.419,A -85,B 0,C 180,E1 -8196.466,E2 -8196.466} C_VEL
LIN {X 0,Y 454.959,Z 308.439,A -85,B 0,C 180,E1 -8198.886,E2 -8198.886} C_VEL
LIN {X 0,Y 454.302,Z 303.088,A -85,B 0,C 180,E1 -8200.022,E2 -8200.022} C_VEL
LIN {X 0,Y 453.578,Z 298.987,A -85,B 0,C 180,E1 -8200.941,E2 -8200.941} C_VEL
LIN {X 0,Y 453.504,Z 298.997,A -85,B 0,C 180,E1 -8203.441,E2 -8203.441} C_VEL
LIN {X 0,Y 453.502,Z 298.995,A -85,B 0,C 180,E1 -8206.197,E2 -8206.197} C_VEL
LIN {X 0,Y 453.518,Z 298.987,A -85,B 0,C 180,E1 -8209.038,E2 -8209.038} C_VEL
LIN {X 0,Y 453.478,Z 298.997,A -85,B 0,C 180,E1 -8211.835,E2 -8211.835} C_VEL
LIN {X 0,Y 453.468,Z 298.996,A -85,B 0,C 180,E1 -8214.736,E2 -8214.736} C_VEL
LIN {X 0,Y 453.46,Z 298.998,A -85,B 0,C 180,E1 -8217.941,E2 -8217.941} C_VEL
LIN {X 0,Y 453.453,Z 299,A -85,B 0,C 180,E1 -8220.76,E2 -8220.76} C_VEL
LIN {X 0,Y 453.464,Z 298.995,A -85,B 0,C 180,E1 -8223.913,E2 -8223.913} C_VEL
LIN {X 0,Y 453.436,Z 299,A -85,B 0,C 180,E1 -8227.19,E2 -8227.19} C_VEL
LIN {X 0,Y 453.466,Z 299.001,A -85,B 0,C 180,E1 -8230.611,E2 -8230.611} C_VEL
LIN {X 0,Y 453.476,Z 298.996,A -85,B 0,C 180,E1 -8234.527,E2 -8234.527} C_VEL
LIN {X 0,Y 453.43,Z 298.998,A -85,B 0,C 180,E1 -8238.07,E2 -8238.07} C_VEL
LIN {X 0,Y 453.436,Z 299.002,A -85,B 0,C 180,E1 -8240.801,E2 -8240.801} C_VEL
LIN {X 0,Y 453.436,Z 298.998,A -85,B 0,C 180,E1 -8243.915,E2 -8243.915} C_VEL
LIN {X 0,Y 453.457,Z 298.998,A -85,B 0,C 180,E1 -8246.815,E2 -8246.815} C_VEL
LIN {X 0,Y 453.44,Z 298.997,A -85,B 0,C 180,E1 -8250.265,E2 -8250.265} C_VEL
LIN {X 0,Y 453.415,Z 299.006,A -85,B 0,C 180,E1 -8253.288,E2 -8253.288} C_VEL
LIN {X 0,Y 453.482,Z 298.993,A -85,B 0,C 180,E1 -8256.237,E2 -8256.237} C_VEL
LIN {X 0,Y 453.472,Z 298.995,A -85,B 0,C 180,E1 -8259.117,E2 -8259.117} C_VEL
LIN {X 0,Y 453.455,Z 299.001,A -85,B 0,C 180,E1 -8261.942,E2 -8261.942} C_VEL
LIN {X 0,Y 453.476,Z 298.993,A -85,B 0,C 180,E1 -8264.724,E2 -8264.724} C_VEL
LIN {X 0,Y 453.555,Z 298.985,A -85,B 0,C 180,E1 -8267.471,E2 -8267.471} C_VEL
LIN {X 0,Y 453.548,Z 298.984,A -85,B 0,C 180,E1 -8271.086,E2 -8271.086} C_VEL
LIN {X 0,Y 453.624,Z 298.978,A -85,B 0,C 180,E1 -8273.774,E2 -8273.774} C_VEL
LIN {X 0,Y 453.703,Z 298.965,A -85,B 0,C 180,E1 -8277.336,E2 -8277.336} C_VEL
LIN {X 0,Y 453.755,Z 298.962,A -85,B 0,C 180,E1 -8280,E2 -8280} C_VEL
LIN {X 0,Y 453.699,Z 298.97,A -85,B 0,C 180,E1 -8282.663,E2 -8282.663} C_VEL
LIN {X 0,Y 453.646,Z 298.976,A -85,B 0,C 180,E1 -8286.226,E2 -8286.226} C_VEL
LIN {X 0,Y 453.568,Z 298.986,A -85,B 0,C 180,E1 -8288.914,E2 -8288.914} C_VEL
LIN {X 0,Y 453.555,Z 298.989,A -85,B 0,C 180,E1 -8292.529,E2 -8292.529} C_VEL
LIN {X 0,Y 453.535,Z 298.986,A -85,B 0,C 180,E1 -8296.196,E2 -8296.196} C_VEL
LIN {X 0,Y 453.508,Z 298.996,A -85,B 0,C 180,E1 -8299.039,E2 -8299.039} C_VEL
LIN {X 0,Y 453.468,Z 298.994,A -85,B 0,C 180,E1 -8301.837,E2 -8301.837} C_VEL
LIN {X 0,Y 453.483,Z 298.995,A -85,B 0,C 180,E1 -8304.736,E2 -8304.736} C_VEL
LIN {X 0,Y 453.521,Z 298.988,A -85,B 0,C 180,E1 -8307.959,E2 -8307.959} C_VEL
LIN {X 0,Y 453.458,Z 299.001,A -85,B 0,C 180,E1 -8311.526,E2 -8311.526} C_VEL
LIN {X 0,Y 453.479,Z 298.993,A -85,B 0,C 180,E1 -8314.778,E2 -8314.778} C_VEL
LIN {X 0,Y 453.451,Z 298.996,A -85,B 0,C 180,E1 -8318.313,E2 -8318.313} C_VEL
LIN {X 0,Y 453.487,Z 298.991,A -85,B 0,C 180,E1 -8320.61,E2 -8320.61} C_VEL
LIN {X 0,Y 453.455,Z 298.998,A -85,B 0,C 180,E1 -8324.223,E2 -8324.223} C_VEL
LIN {X 0,Y 453.443,Z 298.997,A -85,B 0,C 180,E1 -8327.004,E2 -8327.004} C_VEL
LIN {X 0,Y 453.489,Z 298.993,A -85,B 0,C 180,E1 -8329.41,E2 -8329.41} C_VEL
LIN {X 0,Y 453.445,Z 298.997,A -85,B 0,C 180,E1 -8332.811,E2 -8332.811} C_VEL
LIN {X 0,Y 453.473,Z 299.002,A -85,B 0,C 180,E1 -8336.088,E2 -8336.088} C_VEL
LIN {X 0,Y 453.473,Z 298.993,A -85,B 0,C 180,E1 -8339.241,E2 -8339.241} C_VEL
LIN {X 0,Y 453.53,Z 298.994,A -85,B 0,C 180,E1 -8342.298,E2 -8342.298} C_VEL
LIN {X 0,Y 453.512,Z 299.094,A -85,B 0,C 180,E1 -8344.169,E2 -8344.169} C_VEL
LIN {X 0,Y 455.746,Z 311.485,A -85,B 0,C 180,E1 -8346.605,E2 -8346.605} C_VEL
LIN {X 0,Y 454.921,Z 329.47,A -85,B 0,C 180,E1 -8349.896,E2 -8349.896} C_VEL
LIN {X 0,Y 454.315,Z 344.087,A -85,B 0,C 180,E1 -8352.543,E2 -8352.543} C_VEL
LIN {X 0,Y 457.399,Z 364.694,A -85,B 0,C 180,E1 -8352.997,E2 -8352.997} C_VEL
LIN {X 0,Y 456.724,Z 452.848,A -85,B 0,C 180,E1 -8354.408,E2 -8354.408} C_VEL
LIN {X 0,Y 456.229,Z 466.746,A -85,B 0,C 180,E1 -8354.819,E2 -8354.819} C_VEL
LIN {X 0,Y 455.807,Z 479.209,A -85,B 0,C 180,E1 -8355.376,E2 -8355.376} C_VEL
LIN {X 0,Y 455.25,Z 491.92,A -85,B 0,C 180,E1 -8356.157,E2 -8356.157} C_VEL
LIN {X 0,Y 454.679,Z 502.812,A -85,B 0,C 180,E1 -8357.014,E2 -8357.014} C_VEL
LIN {X 0,Y 454.155,Z 513.385,A -85,B 0,C 180,E1 -8358.056,E2 -8358.056} C_VEL
LIN {X 0,Y 453.558,Z 523.365,A -85,B 0,C 180,E1 -8359.285,E2 -8359.285} C_VEL
LIN {X 0,Y 453.167,Z 532.154,A -85,B 0,C 180,E1 -8360.629,E2 -8360.629} C_VEL
LIN {X 0,Y 452.849,Z 539.155,A -85,B 0,C 180,E1 -8361.972,E2 -8361.972} C_VEL
LIN {X 0,Y 452.642,Z 544.761,A -85,B 0,C 180,E1 -8363.314,E2 -8363.314} C_VEL
LIN {X 0,Y 452.564,Z 549.16,A -85,B 0,C 180,E1 -8364.654,E2 -8364.654} C_VEL
LIN {X 0,Y 452.486,Z 551.482,A -85,B 0,C 180,E1 -8365.547,E2 -8365.547} C_VEL
LIN {X 0,Y 452.48,Z 553.375,A -85,B 0,C 180,E1 -8366.439,E2 -8366.439} C_VEL
LIN {X 0,Y 452.507,Z 554.807,A -85,B 0,C 180,E1 -8367.33,E2 -8367.33} C_VEL
LIN {X 0,Y 452.428,Z 556.445,A -85,B 0,C 180,E1 -8369.111,E2 -8369.111} C_VEL
LIN {X 0,Y 452.435,Z 556.683,A -85,B 0,C 180,E1 -8370.001,E2 -8370.001} C_VEL
LIN {X 0,Y 452.428,Z 556.496,A -85,B 0,C 180,E1 -8370.891,E2 -8370.891} C_VEL
LIN {X 0,Y 452.507,Z 554.926,A -85,B 0,C 180,E1 -8372.671,E2 -8372.671} C_VEL
LIN {X 0,Y 452.48,Z 553.552,A -85,B 0,C 180,E1 -8373.563,E2 -8373.563} C_VEL
LIN {X 0,Y 452.545,Z 550.652,A -85,B 0,C 180,E1 -8374.9,E2 -8374.9} C_VEL
LIN {X 0,Y 452.611,Z 546.212,A -85,B 0,C 180,E1 -8376.396,E2 -8376.396} C_VEL
LIN {X 0,Y 452.805,Z 541.674,A -85,B 0,C 180,E1 -8377.582,E2 -8377.582} C_VEL
LIN {X 0,Y 453.085,Z 535.335,A -85,B 0,C 180,E1 -8378.924,E2 -8378.924} C_VEL
LIN {X 0,Y 453.482,Z 527.409,A -85,B 0,C 180,E1 -8380.267,E2 -8380.267} C_VEL
LIN {X 0,Y 453.982,Z 519.351,A -85,B 0,C 180,E1 -8381.384,E2 -8381.384} C_VEL
LIN {X 0,Y 454.545,Z 509.537,A -85,B 0,C 180,E1 -8382.502,E2 -8382.502} C_VEL
LIN {X 0,Y 455.097,Z 498.586,A -85,B 0,C 180,E1 -8383.508,E2 -8383.508} C_VEL
LIN {X 0,Y 455.76,Z 486.105,A -85,B 0,C 180,E1 -8384.398,E2 -8384.398} C_VEL
LIN {X 0,Y 456.368,Z 473.835,A -85,B 0,C 180,E1 -8385.063,E2 -8385.063} C_VEL
LIN {X 0,Y 456.849,Z 460.857,A -85,B 0,C 180,E1 -8385.561,E2 -8385.561} C_VEL
LIN {X 0,Y 457.158,Z 447.021,A -85,B 0,C 180,E1 -8385.893,E2 -8385.893} C_VEL
LIN {X 0,Y 457.903,Z 364.372,A -85,B 0,C 180,E1 -8387.208,E2 -8387.208} C_VEL
LIN {X 0,Y 454.505,Z 343.934,A -85,B 0,C 180,E1 -8387.701,E2 -8387.701} C_VEL
LIN {X 0,Y 455.301,Z 327.067,A -85,B 0,C 180,E1 -8390.796,E2 -8390.796} C_VEL
LIN {X 0,Y 456.059,Z 313.179,A -85,B 0,C 180,E1 -8393.38,E2 -8393.38} C_VEL
LIN {X 0,Y 455.13,Z 306.871,A -85,B 0,C 180,E1 -8394.641,E2 -8394.641} C_VEL
LIN {X 0,Y 453.501,Z 298.999,A -85,B 0,C 180,E1 -8396.31,E2 -8396.31} C_VEL
LIN {X 0,Y 453.51,Z 298.998,A -85,B 0,C 180,E1 -8398.712,E2 -8398.712} C_VEL
LIN {X 0,Y 453.467,Z 299.003,A -85,B 0,C 180,E1 -8401.8,E2 -8401.8} C_VEL
LIN {X 0,Y 453.481,Z 298.997,A -85,B 0,C 180,E1 -8404.99,E2 -8404.99} C_VEL
LIN {X 0,Y 453.459,Z 299.003,A -85,B 0,C 180,E1 -8408.312,E2 -8408.312} C_VEL
LIN {X 0,Y 453.495,Z 298.995,A -85,B 0,C 180,E1 -8410.609,E2 -8410.609} C_VEL
LIN {X 0,Y 453.461,Z 299.001,A -85,B 0,C 180,E1 -8414.222,E2 -8414.222} C_VEL
LIN {X 0,Y 453.45,Z 299,A -85,B 0,C 180,E1 -8417.003,E2 -8417.003} C_VEL
LIN {X 0,Y 453.495,Z 298.991,A -85,B 0,C 180,E1 -8419.409,E2 -8419.409} C_VEL
LIN {X 0,Y 453.451,Z 299.003,A -85,B 0,C 180,E1 -8422.81,E2 -8422.81} C_VEL
LIN {X 0,Y 453.477,Z 298.994,A -85,B 0,C 180,E1 -8426.087,E2 -8426.087} C_VEL
LIN {X 0,Y 453.476,Z 298.998,A -85,B 0,C 180,E1 -8429.24,E2 -8429.24} C_VEL
LIN {X 0,Y 453.508,Z 298.988,A -85,B 0,C 180,E1 -8432.296,E2 -8432.296} C_VEL
LIN {X 0,Y 453.494,Z 298.995,A -85,B 0,C 180,E1 -8435.264,E2 -8435.264} C_VEL
LIN {X 0,Y 453.481,Z 298.992,A -85,B 0,C 180,E1 -8438.415,E2 -8438.415} C_VEL
LIN {X 0,Y 453.523,Z 298.99,A -85,B 0,C 180,E1 -8441.009,E2 -8441.009} C_VEL
LIN {X 0,Y 453.57,Z 298.983,A -85,B 0,C 180,E1 -8443.88,E2 -8443.88} C_VEL
LIN {X 0,Y 453.565,Z 298.984,A -85,B 0,C 180,E1 -8447.471,E2 -8447.471} C_VEL
LIN {X 0,Y 453.585,Z 298.978,A -85,B 0,C 180,E1 -8451.087,E2 -8451.087} C_VEL
LIN {X 0,Y 453.665,Z 298.974,A -85,B 0,C 180,E1 -8453.775,E2 -8453.775} C_VEL
LIN {X 0,Y 453.732,Z 298.959,A -85,B 0,C 180,E1 -8457.337,E2 -8457.337} C_VEL
LIN {X 0,Y 453.82,Z 298.953,A -85,B 0,C 180,E1 -8460,E2 -8460} C_VEL
LIN {X 0,Y 453.735,Z 298.962,A -85,B 0,C 180,E1 -8462.664,E2 -8462.664} C_VEL
LIN {X 0,Y 453.652,Z 298.975,A -85,B 0,C 180,E1 -8466.226,E2 -8466.226} C_VEL
LIN {X 0,Y 453.587,Z 298.978,A -85,B 0,C 180,E1 -8468.914,E2 -8468.914} C_VEL
LIN {X 0,Y 453.565,Z 298.987,A -85,B 0,C 180,E1 -8472.529,E2 -8472.529} C_VEL
LIN {X 0,Y 453.546,Z 298.987,A -85,B 0,C 180,E1 -8476.196,E2 -8476.196} C_VEL
LIN {X 0,Y 453.519,Z 298.993,A -85,B 0,C 180,E1 -8479.04,E2 -8479.04} C_VEL
LIN {X 0,Y 453.478,Z 298.99,A -85,B 0,C 180,E1 -8481.836,E2 -8481.836} C_VEL
LIN {X 0,Y 453.502,Z 298.994,A -85,B 0,C 180,E1 -8484.735,E2 -8484.735} C_VEL
LIN {X 0,Y 453.508,Z 298.987,A -85,B 0,C 180,E1 -8487.953,E2 -8487.953} C_VEL
LIN {X 0,Y 453.477,Z 298.995,A -85,B 0,C 180,E1 -8490.76,E2 -8490.76} C_VEL
LIN {X 0,Y 453.47,Z 298.994,A -85,B 0,C 180,E1 -8493.914,E2 -8493.914} C_VEL
LIN {X 0,Y 453.452,Z 299.001,A -85,B 0,C 180,E1 -8497.19,E2 -8497.19} C_VEL
LIN {X 0,Y 453.496,Z 298.992,A -85,B 0,C 180,E1 -8500.609,E2 -8500.609} C_VEL
LIN {X 0,Y 453.464,Z 299,A -85,B 0,C 180,E1 -8504.222,E2 -8504.222} C_VEL
LIN {X 0,Y 453.44,Z 299.001,A -85,B 0,C 180,E1 -8507.002,E2 -8507.002} C_VEL
LIN {X 0,Y 453.474,Z 298.998,A -85,B 0,C 180,E1 -8509.413,E2 -8509.413} C_VEL
LIN {X 0,Y 453.452,Z 299.002,A -85,B 0,C 180,E1 -8512.81,E2 -8512.81} C_VEL
LIN {X 0,Y 453.471,Z 299,A -85,B 0,C 180,E1 -8516.086,E2 -8516.086} C_VEL
LIN {X 0,Y 453.49,Z 299.007,A -85,B 0,C 180,E1 -8516.937,E2 -8516.937} C_VEL
LIN {X 0,Y 454.924,Z 306.556,A -85,B 0,C 180,E1 -8518.574,E2 -8518.574} C_VEL
LIN {X 0,Y 454.79,Z 316.654,A -85,B 0,C 180,E1 -8520.617,E2 -8520.617} C_VEL
LIN {X 0,Y 454.713,Z 320.58,A -85,B 0,C 180,E1 -8521.365,E2 -8521.365} C_VEL
LIN {X 0,Y 458.09,Z 337.154,A -85,B 0,C 180,E1 -8521.789,E2 -8521.789} C_VEL
LIN {X 0,Y 457.197,Z 427.807,A -85,B 0,C 180,E1 -8523.249,E2 -8523.249} C_VEL
LIN {X 0,Y 456.885,Z 440.417,A -85,B 0,C 180,E1 -8523.618,E2 -8523.618} C_VEL
LIN {X 0,Y 456.442,Z 452.814,A -85,B 0,C 180,E1 -8524.155,E2 -8524.155} C_VEL
LIN {X 0,Y 456.161,Z 459.237,A -85,B 0,C 180,E1 -8524.506,E2 -8524.506} C_VEL
LIN {X 0,Y 455.316,Z 464.598,A -85,B 0,C 180,E1 -8524.821,E2 -8524.821} C_VEL
LIN {X 0,Y 452.09,Z 472.999,A -85,B 0,C 180,E1 -8525.339,E2 -8525.339} C_VEL
LIN {X 0,Y 448.825,Z 481.069,A -85,B 0,C 180,E1 -8525.943,E2 -8525.943} C_VEL
LIN {X 0,Y 447.919,Z 485.698,A -85,B 0,C 180,E1 -8526.392,E2 -8526.392} C_VEL
LIN {X 0,Y 447.273,Z 495.909,A -85,B 0,C 180,E1 -8527.601,E2 -8527.601} C_VEL
LIN {X 0,Y 446.783,Z 504.023,A -85,B 0,C 180,E1 -8528.789,E2 -8528.789} C_VEL
LIN {X 0,Y 446.256,Z 511.843,A -85,B 0,C 180,E1 -8530.208,E2 -8530.208} C_VEL
LIN {X 0,Y 445.941,Z 518.074,A -85,B 0,C 180,E1 -8531.627,E2 -8531.627} C_VEL
LIN {X 0,Y 445.665,Z 522.949,A -85,B 0,C 180,E1 -8533.037,E2 -8533.037} C_VEL
LIN {X 0,Y 445.533,Z 526.636,A -85,B 0,C 180,E1 -8534.444,E2 -8534.444} C_VEL
LIN {X 0,Y 445.412,Z 528.507,A -85,B 0,C 180,E1 -8535.376,E2 -8535.376} C_VEL
LIN {X 0,Y 445.335,Z 529.891,A -85,B 0,C 180,E1 -8536.306,E2 -8536.306} C_VEL
LIN {X 0,Y 445.379,Z 531.384,A -85,B 0,C 180,E1 -8538.058,E2 -8538.058} C_VEL
LIN {X 0,Y 445.314,Z 531.576,A -85,B 0,C 180,E1 -8539.083,E2 -8539.083} C_VEL
LIN {X 0,Y 445.31,Z 530.635,A -85,B 0,C 180,E1 -8540.919,E2 -8540.919} C_VEL
LIN {X 0,Y 445.352,Z 529.576,A -85,B 0,C 180,E1 -8541.834,E2 -8541.834} C_VEL
LIN {X 0,Y 445.44,Z 528.063,A -85,B 0,C 180,E1 -8542.748,E2 -8542.748} C_VEL
LIN {X 0,Y 445.531,Z 525.585,A -85,B 0,C 180,E1 -8543.892,E2 -8543.892} C_VEL
LIN {X 0,Y 445.665,Z 520.921,A -85,B 0,C 180,E1 -8545.477,E2 -8545.477} C_VEL
LIN {X 0,Y 445.924,Z 514.664,A -85,B 0,C 180,E1 -8547.063,E2 -8547.063} C_VEL
LIN {X 0,Y 446.264,Z 507.865,A -85,B 0,C 180,E1 -8548.42,E2 -8548.42} C_VEL
LIN {X 0,Y 446.744,Z 500.919,A -85,B 0,C 180,E1 -8549.549,E2 -8549.549} C_VEL
LIN {X 0,Y 447.079,Z 492.612,A -85,B 0,C 180,E1 -8550.675,E2 -8550.675} C_VEL
LIN {X 0,Y 447.654,Z 483.493,A -85,B 0,C 180,E1 -8551.686,E2 -8551.686} C_VEL
LIN {X 0,Y 448.258,Z 473.575,A -85,B 0,C 180,E1 -8552.583,E2 -8552.583} C_VEL
LIN {X 0,Y 448.834,Z 461.094,A -85,B 0,C 180,E1 -8553.478,E2 -8553.478} C_VEL
LIN {X 0,Y 449.25,Z 448.764,A -85,B 0,C 180,E1 -8554.148,E2 -8554.148} C_VEL
LIN {X 0,Y 449.594,Z 435.611,A -85,B 0,C 180,E1 -8554.651,E2 -8554.651} C_VEL
LIN {X 0,Y 449.895,Z 422.755,A -85,B 0,C 180,E1 -8554.956,E2 -8554.956} C_VEL
LIN {X 0,Y 450.623,Z 337.291,A -85,B 0,C 180,E1 -8556.323,E2 -8556.323} C_VEL
LIN {X 0,Y 447.384,Z 320.485,A -85,B 0,C 180,E1 -8556.737,E2 -8556.737} C_VEL
LIN {X 0,Y 447.986,Z 309.286,A -85,B 0,C 180,E1 -8559.025,E2 -8559.025} C_VEL
LIN {X 0,Y 446.867,Z 301.78,A -85,B 0,C 180,E1 -8560.648,E2 -8560.648} C_VEL
LIN {X 0,Y 446.543,Z 299.864,A -85,B 0,C 180,E1 -8561.115,E2 -8561.115} C_VEL
LIN {X 0,Y 446.463,Z 299.874,A -85,B 0,C 180,E1 -8563.657,E2 -8563.657} C_VEL
LIN {X 0,Y 446.443,Z 299.871,A -85,B 0,C 180,E1 -8566.46,E2 -8566.46} C_VEL
LIN {X 0,Y 446.47,Z 299.866,A -85,B 0,C 180,E1 -8569.302,E2 -8569.302} C_VEL
LIN {X 0,Y 446.419,Z 299.88,A -85,B 0,C 180,E1 -8572.199,E2 -8572.199} C_VEL
LIN {X 0,Y 446.419,Z 299.872,A -85,B 0,C 180,E1 -8575.154,E2 -8575.154} C_VEL
LIN {X 0,Y 446.416,Z 299.878,A -85,B 0,C 180,E1 -8578.182,E2 -8578.182} C_VEL
LIN {X 0,Y 446.405,Z 299.874,A -85,B 0,C 180,E1 -8581.3,E2 -8581.3} C_VEL
LIN {X 0,Y 446.42,Z 299.88,A -85,B 0,C 180,E1 -8584.523,E2 -8584.523} C_VEL
LIN {X 0,Y 446.399,Z 299.876,A -85,B 0,C 180,E1 -8588.076,E2 -8588.076} C_VEL
LIN {X 0,Y 446.396,Z 299.876,A -85,B 0,C 180,E1 -8591.393,E2 -8591.393} C_VEL
LIN {X 0,Y 446.444,Z 299.874,A -85,B 0,C 180,E1 -8595.103,E2 -8595.103} C_VEL
LIN {X 0,Y 446.394,Z 299.878,A -85,B 0,C 180,E1 -8598.605,E2 -8598.605} C_VEL
LIN {X 0,Y 446.394,Z 299.875,A -85,B 0,C 180,E1 -8601.922,E2 -8601.922} C_VEL
LIN {X 0,Y 446.407,Z 299.878,A -85,B 0,C 180,E1 -8605.475,E2 -8605.475} C_VEL
LIN {X 0,Y 446.38,Z 299.878,A -85,B 0,C 180,E1 -8608.696,E2 -8608.696} C_VEL
LIN {X 0,Y 446.393,Z 299.878,A -85,B 0,C 180,E1 -8611.841,E2 -8611.841} C_VEL
LIN {X 0,Y 446.404,Z 299.875,A -85,B 0,C 180,E1 -8614.844,E2 -8614.844} C_VEL
LIN {X 0,Y 446.44,Z 299.871,A -85,B 0,C 180,E1 -8618.245,E2 -8618.245} C_VEL
LIN {X 0,Y 446.411,Z 299.88,A -85,B 0,C 180,E1 -8621.647,E2 -8621.647} C_VEL
LIN {X 0,Y 446.419,Z 299.873,A -85,B 0,C 180,E1 -8624.476,E2 -8624.476} C_VEL
LIN {X 0,Y 446.507,Z 299.863,A -85,B 0,C 180,E1 -8627.384,E2 -8627.384} C_VEL
LIN {X 0,Y 446.499,Z 299.862,A -85,B 0,C 180,E1 -8630.944,E2 -8630.944} C_VEL
LIN {X 0,Y 446.594,Z 299.853,A -85,B 0,C 180,E1 -8633.675,E2 -8633.675} C_VEL
LIN {X 0,Y 446.652,Z 299.843,A -85,B 0,C 180,E1 -8637.294,E2 -8637.294} C_VEL
LIN {X 0,Y 446.706,Z 299.84,A -85,B 0,C 180,E1 -8640,E2 -8640} C_VEL
LIN {X 0,Y 446.648,Z 299.848,A -85,B 0,C 180,E1 -8642.705,E2 -8642.705} C_VEL
LIN {X 0,Y 446.615,Z 299.853,A -85,B 0,C 180,E1 -8646.324,E2 -8646.324} C_VEL
LIN {X 0,Y 446.516,Z 299.863,A -85,B 0,C 180,E1 -8649.056,E2 -8649.056} C_VEL
LIN {X 0,Y 446.512,Z 299.869,A -85,B 0,C 180,E1 -8652.73,E2 -8652.73} C_VEL
LIN {X 0,Y 446.479,Z 299.868,A -85,B 0,C 180,E1 -8656.459,E2 -8656.459} C_VEL
LIN {X 0,Y 446.459,Z 299.871,A -85,B 0,C 180,E1 -8659.304,E2 -8659.304} C_VEL
LIN {X 0,Y 446.409,Z 299.873,A -85,B 0,C 180,E1 -8662.2,E2 -8662.2} C_VEL
LIN {X 0,Y 446.428,Z 299.879,A -85,B 0,C 180,E1 -8665.154,E2 -8665.154} C_VEL
LIN {X 0,Y 446.477,Z 299.865,A -85,B 0,C 180,E1 -8668.179,E2 -8668.179} C_VEL
LIN {X 0,Y 446.411,Z 299.876,A -85,B 0,C 180,E1 -8671.775,E2 -8671.775} C_VEL
LIN {X 0,Y 446.421,Z 299.872,A -85,B 0,C 180,E1 -8674.524,E2 -8674.524} C_VEL
LIN {X 0,Y 446.404,Z 299.876,A -85,B 0,C 180,E1 -8678.079,E2 -8678.079} C_VEL
LIN {X 0,Y 446.412,Z 299.878,A -85,B 0,C 180,E1 -8681.393,E2 -8681.393} C_VEL
LIN {X 0,Y 446.444,Z 299.87,A -85,B 0,C 180,E1 -8685.105,E2 -8685.105} C_VEL
LIN {X 0,Y 446.413,Z 299.873,A -85,B 0,C 180,E1 -8688.609,E2 -8688.609} C_VEL
LIN {X 0,Y 446.419,Z 299.872,A -85,B 0,C 180,E1 -8690.972,E2 -8690.972} C_VEL
LIN {X 0,Y 446.414,Z 299.877,A -85,B 0,C 180,E1 -8694.375,E2 -8694.375} C_VEL
LIN {X 0,Y 446.419,Z 299.874,A -85,B 0,C 180,E1 -8697.639,E2 -8697.639} C_VEL
LIN {X 0,Y 446.445,Z 299.872,A -85,B 0,C 180,E1 -8700.791,E2 -8700.791} C_VEL
LIN {X 0,Y 446.455,Z 299.926,A -85,B 0,C 180,E1 -8703.974,E2 -8703.974} C_VEL
LIN {X 0,Y 448.75,Z 312.369,A -85,B 0,C 180,E1 -8706.463,E2 -8706.463} C_VEL
LIN {X 0,Y 448.014,Z 329.09,A -85,B 0,C 180,E1 -8709.573,E2 -8709.573} C_VEL
LIN {X 0,Y 447.33,Z 344.052,A -85,B 0,C 180,E1 -8712.314,E2 -8712.314} C_VEL
LIN {X 0,Y 450.565,Z 366.302,A -85,B 0,C 180,E1 -8712.79,E2 -8712.79} C_VEL
LIN {X 0,Y 449.826,Z 452.662,A -85,B 0,C 180,E1 -8714.191,E2 -8714.191} C_VEL
LIN {X 0,Y 449.351,Z 466.564,A -85,B 0,C 180,E1 -8714.61,E2 -8714.61} C_VEL
LIN {X 0,Y 448.861,Z 479.534,A -85,B 0,C 180,E1 -8715.203,E2 -8715.203} C_VEL
LIN {X 0,Y 448.317,Z 491.337,A -85,B 0,C 180,E1 -8715.938,E2 -8715.938} C_VEL
LIN {X 0,Y 447.657,Z 503.448,A -85,B 0,C 180,E1 -8716.908,E2 -8716.908} C_VEL
LIN {X 0,Y 447.11,Z 513.941,A -85,B 0,C 180,E1 -8717.98,E2 -8717.98} C_VEL
LIN {X 0,Y 446.548,Z 522.98,A -85,B 0,C 180,E1 -8719.114,E2 -8719.114} C_VEL
LIN {X 0,Y 446.125,Z 531.808,A -85,B 0,C 180,E1 -8720.48,E2 -8720.48} C_VEL
LIN {X 0,Y 445.787,Z 538.847,A -85,B 0,C 180,E1 -8721.844,E2 -8721.844} C_VEL
LIN {X 0,Y 445.576,Z 544.477,A -85,B 0,C 180,E1 -8723.207,E2 -8723.207} C_VEL
LIN {X 0,Y 445.478,Z 548.897,A -85,B 0,C 180,E1 -8724.569,E2 -8724.569} C_VEL
LIN {X 0,Y 445.411,Z 551.229,A -85,B 0,C 180,E1 -8725.476,E2 -8725.476} C_VEL
LIN {X 0,Y 445.379,Z 553.131,A -85,B 0,C 180,E1 -8726.382,E2 -8726.382} C_VEL
LIN {X 0,Y 445.432,Z 554.58,A -85,B 0,C 180,E1 -8727.288,E2 -8727.288} C_VEL
LIN {X 0,Y 445.338,Z 556.234,A -85,B 0,C 180,E1 -8729.096,E2 -8729.096} C_VEL
LIN {X 0,Y 445.342,Z 556.481,A -85,B 0,C 180,E1 -8730.001,E2 -8730.001} C_VEL
LIN {X 0,Y 445.338,Z 556.309,A -85,B 0,C 180,E1 -8730.905,E2 -8730.905} C_VEL
LIN {X 0,Y 445.432,Z 554.756,A -85,B 0,C 180,E1 -8732.714,E2 -8732.714} C_VEL
LIN {X 0,Y 445.378,Z 553.39,A -85,B 0,C 180,E1 -8733.62,E2 -8733.62} C_VEL
LIN {X 0,Y 445.474,Z 550.508,A -85,B 0,C 180,E1 -8734.978,E2 -8734.978} C_VEL
LIN {X 0,Y 445.53,Z 546.456,A -85,B 0,C 180,E1 -8736.386,E2 -8736.386} C_VEL
LIN {X 0,Y 445.733,Z 541.572,A -85,B 0,C 180,E1 -8737.703,E2 -8737.703} C_VEL
LIN {X 0,Y 446.021,Z 535.266,A -85,B 0,C 180,E1 -8739.067,E2 -8739.067} C_VEL
LIN {X 0,Y 446.469,Z 527.379,A -85,B 0,C 180,E1 -8740.43,E2 -8740.43} C_VEL
LIN {X 0,Y 447.022,Z 519.359,A -85,B 0,C 180,E1 -8741.564,E2 -8741.564} C_VEL
LIN {X 0,Y 447.593,Z 509.594,A -85,B 0,C 180,E1 -8742.699,E2 -8742.699} C_VEL
LIN {X 0,Y 448.199,Z 498.73,A -85,B 0,C 180,E1 -8743.72,E2 -8743.72} C_VEL
LIN {X 0,Y 448.905,Z 486.348,A -85,B 0,C 180,E1 -8744.623,E2 -8744.623} C_VEL
LIN {X 0,Y 449.548,Z 474.215,A -85,B 0,C 180,E1 -8745.297,E2 -8745.297} C_VEL
LIN {X 0,Y 450.059,Z 461.596,A -85,B 0,C 180,E1 -8745.802,E2 -8745.802} C_VEL
LIN {X 0,Y 450.375,Z 448.378,A -85,B 0,C 180,E1 -8746.139,E2 -8746.139} C_VEL
LIN {X 0,Y 451.099,Z 364.586,A -85,B 0,C 180,E1 -8747.502,E2 -8747.502} C_VEL
LIN {X 0,Y 447.569,Z 343.626,A -85,B 0,C 180,E1 -8748.038,E2 -8748.038} C_VEL
LIN {X 0,Y 448.516,Z 325.795,A -85,B 0,C 180,E1 -8751.366,E2 -8751.366} C_VEL
LIN {X 0,Y 449.16,Z 314.443,A -85,B 0,C 180,E1 -8753.516,E2 -8753.516} C_VEL
LIN {X 0,Y 448.209,Z 308.365,A -85,B 0,C 180,E1 -8754.756,E2 -8754.756} C_VEL
LIN {X 0,Y 446.448,Z 299.877,A -85,B 0,C 180,E1 -8756.588,E2 -8756.588} C_VEL
LIN {X 0,Y 446.45,Z 299.88,A -85,B 0,C 180,E1 -8759.21,E2 -8759.21} C_VEL
LIN {X 0,Y 446.425,Z 299.877,A -85,B 0,C 180,E1 -8762.362,E2 -8762.362} C_VEL
LIN {X 0,Y 446.42,Z 299.88,A -85,B 0,C 180,E1 -8765.626,E2 -8765.626} C_VEL
LIN {X 0,Y 446.411,Z 299.875,A -85,B 0,C 180,E1 -8769.031,E2 -8769.031} C_VEL
LIN {X 0,Y 446.423,Z 299.879,A -85,B 0,C 180,E1 -8772.276,E2 -8772.276} C_VEL
LIN {X 0,Y 446.452,Z 299.87,A -85,B 0,C 180,E1 -8775.104,E2 -8775.104} C_VEL
LIN {X 0,Y 446.42,Z 299.877,A -85,B 0,C 180,E1 -8778.608,E2 -8778.608} C_VEL
LIN {X 0,Y 446.412,Z 299.871,A -85,B 0,C 180,E1 -8781.922,E2 -8781.922} C_VEL
LIN {X 0,Y 446.429,Z 299.872,A -85,B 0,C 180,E1 -8785.477,E2 -8785.477} C_VEL
LIN {X 0,Y 446.416,Z 299.875,A -85,B 0,C 180,E1 -8788.7,E2 -8788.7} C_VEL
LIN {X 0,Y 446.451,Z 299.867,A -85,B 0,C 180,E1 -8791.83,E2 -8791.83} C_VEL
LIN {X 0,Y 446.439,Z 299.875,A -85,B 0,C 180,E1 -8794.847,E2 -8794.847} C_VEL
LIN {X 0,Y 446.449,Z 299.868,A -85,B 0,C 180,E1 -8798.245,E2 -8798.245} C_VEL
LIN {X 0,Y 446.453,Z 299.871,A -85,B 0,C 180,E1 -8801.649,E2 -8801.649} C_VEL
LIN {X 0,Y 446.508,Z 299.86,A -85,B 0,C 180,E1 -8804.48,E2 -8804.48} C_VEL
LIN {X 0,Y 446.518,Z 299.859,A -85,B 0,C 180,E1 -8808.193,E2 -8808.193} C_VEL
LIN {X 0,Y 446.532,Z 299.855,A -85,B 0,C 180,E1 -8810.945,E2 -8810.945} C_VEL
LIN {X 0,Y 446.634,Z 299.848,A -85,B 0,C 180,E1 -8813.676,E2 -8813.676} C_VEL
LIN {X 0,Y 446.679,Z 299.837,A -85,B 0,C 180,E1 -8817.295,E2 -8817.295} C_VEL
LIN {X 0,Y 446.79,Z 299.828,A -85,B 0,C 180,E1 -8820,E2 -8820} C_VEL
LIN {X 0,Y 446.682,Z 299.84,A -85,B 0,C 180,E1 -8822.706,E2 -8822.706} C_VEL
LIN {X 0,Y 446.62,Z 299.852,A -85,B 0,C 180,E1 -8826.324,E2 -8826.324} C_VEL
LIN {X 0,Y 446.522,Z 299.858,A -85,B 0,C 180,E1 -8829.97,E2 -8829.97} C_VEL
LIN {X 0,Y 446.523,Z 299.861,A -85,B 0,C 180,E1 -8832.73,E2 -8832.73} C_VEL
LIN {X 0,Y 446.498,Z 299.866,A -85,B 0,C 180,E1 -8836.228,E2 -8836.228} C_VEL
LIN {X 0,Y 446.47,Z 299.868,A -85,B 0,C 180,E1 -8839.303,E2 -8839.303} C_VEL
LIN {X 0,Y 446.419,Z 299.87,A -85,B 0,C 180,E1 -8842.2,E2 -8842.2} C_VEL
LIN {X 0,Y 446.444,Z 299.872,A -85,B 0,C 180,E1 -8845.153,E2 -8845.153} C_VEL
LIN {X 0,Y 446.451,Z 299.866,A -85,B 0,C 180,E1 -8848.181,E2 -8848.181} C_VEL
LIN {X 0,Y 446.417,Z 299.877,A -85,B 0,C 180,E1 -8851.301,E2 -8851.301} C_VEL
LIN {X 0,Y 446.425,Z 299.87,A -85,B 0,C 180,E1 -8854.524,E2 -8854.524} C_VEL
LIN {X 0,Y 446.414,Z 299.876,A -85,B 0,C 180,E1 -8858.079,E2 -8858.079} C_VEL
LIN {X 0,Y 446.425,Z 299.874,A -85,B 0,C 180,E1 -8860.917,E2 -8860.917} C_VEL
LIN {X 0,Y 446.402,Z 299.881,A -85,B 0,C 180,E1 -8863.846,E2 -8863.846} C_VEL
LIN {X 0,Y 446.396,Z 299.88,A -85,B 0,C 180,E1 -8866.404,E2 -8866.404} C_VEL
LIN {X 0,Y 446.403,Z 299.878,A -85,B 0,C 180,E1 -8869.797,E2 -8869.797} C_VEL
LIN {X 0,Y 446.407,Z 299.879,A -85,B 0,C 180,E1 -8872.121,E2 -8872.121} C_VEL
LIN {X 0,Y 446.426,Z 299.877,A -85,B 0,C 180,E1 -8875.476,E2 -8875.476} C_VEL
LIN {X 0,Y 446.461,Z 299.977,A -85,B 0,C 180,E1 -8876.702,E2 -8876.702} C_VEL
LIN {X 0,Y 448.069,Z 308.496,A -85,B 0,C 180,E1 -8878.578,E2 -8878.578} C_VEL
LIN {X 0,Y 447.79,Z 320.534,A -85,B 0,C 180,E1 -8881.038,E2 -8881.038} C_VEL
LIN {X 0,Y 451.347,Z 337.917,A -85,B 0,C 180,E1 -8881.499,E2 -8881.499} C_VEL
LIN {X 0,Y 450.431,Z 428.513,A -85,B 0,C 180,E1 -8882.988,E2 -8882.988} C_VEL
LIN {X 0,Y 450.107,Z 440.832,A -85,B 0,C 180,E1 -8883.357,E2 -8883.357} C_VEL
LIN {X 0,Y 449.619,Z 453.533,A -85,B 0,C 180,E1 -8883.92,E2 -8883.92} C_VEL
LIN {X 0,Y 449.144,Z 465.368,A -85,B 0,C 180,E1 -8884.637,E2 -8884.637} C_VEL
LIN {X 0,Y 448.548,Z 475.833,A -85,B 0,C 180,E1 -8885.447,E2 -8885.447} C_VEL
LIN {X 0,Y 447.919,Z 485.698,A -85,B 0,C 180,E1 -8886.392,E2 -8886.392} C_VEL
LIN {X 0,Y 447.012,Z 490.242,A -85,B 0,C 180,E1 -8886.873,E2 -8886.873} C_VEL
LIN {X 0,Y 443.703,Z 497.305,A -85,B 0,C 180,E1 -8887.672,E2 -8887.672} C_VEL
LIN {X 0,Y 440.45,Z 503.795,A -85,B 0,C 180,E1 -8888.545,E2 -8888.545} C_VEL
LIN {X 0,Y 439.625,Z 507.372,A -85,B 0,C 180,E1 -8889.136,E2 -8889.136} C_VEL
LIN {X 0,Y 439.229,Z 513.614,A -85,B 0,C 180,E1 -8890.365,E2 -8890.365} C_VEL
LIN {X 0,Y 438.834,Z 519.507,A -85,B 0,C 180,E1 -8891.802,E2 -8891.802} C_VEL
LIN {X 0,Y 438.555,Z 524.086,A -85,B 0,C 180,E1 -8893.234,E2 -8893.234} C_VEL
LIN {X 0,Y 438.485,Z 526.485,A -85,B 0,C 180,E1 -8894.188,E2 -8894.188} C_VEL
LIN {X 0,Y 438.362,Z 528.43,A -85,B 0,C 180,E1 -8895.136,E2 -8895.136} C_VEL
LIN {X 0,Y 438.251,Z 529.906,A -85,B 0,C 180,E1 -8896.081,E2 -8896.081} C_VEL
LIN {X 0,Y 438.299,Z 531.559,A -85,B 0,C 180,E1 -8897.968,E2 -8897.968} C_VEL
LIN {X 0,Y 438.232,Z 531.79,A -85,B 0,C 180,E1 -8898.904,E2 -8898.904} C_VEL
LIN {X 0,Y 438.214,Z 531.578,A -85,B 0,C 180,E1 -8899.838,E2 -8899.838} C_VEL
LIN {X 0,Y 438.263,Z 529.959,A -85,B 0,C 180,E1 -8901.701,E2 -8901.701} C_VEL
LIN {X 0,Y 438.327,Z 528.549,A -85,B 0,C 180,E1 -8902.63,E2 -8902.63} C_VEL
LIN {X 0,Y 438.439,Z 525.835,A -85,B 0,C 180,E1 -8903.92,E2 -8903.92} C_VEL
LIN {X 0,Y 438.567,Z 521.625,A -85,B 0,C 180,E1 -8905.404,E2 -8905.404} C_VEL
LIN {X 0,Y 438.846,Z 516.5,A -85,B 0,C 180,E1 -8906.786,E2 -8906.786} C_VEL
LIN {X 0,Y 439.093,Z 510.073,A -85,B 0,C 180,E1 -8908.165,E2 -8908.165} C_VEL
LIN {X 0,Y 439.665,Z 502.059,A -85,B 0,C 180,E1 -8909.541,E2 -8909.541} C_VEL
LIN {X 0,Y 440.028,Z 493.932,A -85,B 0,C 180,E1 -8910.686,E2 -8910.686} C_VEL
LIN {X 0,Y 440.621,Z 485.057,A -85,B 0,C 180,E1 -8911.713,E2 -8911.713} C_VEL
LIN {X 0,Y 441.22,Z 475.485,A -85,B 0,C 180,E1 -8912.624,E2 -8912.624} C_VEL
LIN {X 0,Y 441.732,Z 465.216,A -85,B 0,C 180,E1 -8913.42,E2 -8913.42} C_VEL
LIN {X 0,Y 442.218,Z 452.949,A -85,B 0,C 180,E1 -8914.157,E2 -8914.157} C_VEL
LIN {X 0,Y 442.59,Z 440.072,A -85,B 0,C 180,E1 -8914.724,E2 -8914.724} C_VEL
LIN {X 0,Y 442.891,Z 427.483,A -85,B 0,C 180,E1 -8915.092,E2 -8915.092} C_VEL
LIN {X 0,Y 443.919,Z 339.025,A -85,B 0,C 180,E1 -8916.533,E2 -8916.533} C_VEL
LIN {X 0,Y 440.459,Z 320.665,A -85,B 0,C 180,E1 -8916.987,E2 -8916.987} C_VEL
LIN {X 0,Y 440.996,Z 310.139,A -85,B 0,C 180,E1 -8919.169,E2 -8919.169} C_VEL
LIN {X 0,Y 439.506,Z 300.742,A -85,B 0,C 180,E1 -8921.237,E2 -8921.237} C_VEL
LIN {X 0,Y 439.42,Z 300.752,A -85,B 0,C 180,E1 -8923.88,E2 -8923.88} C_VEL
LIN {X 0,Y 439.389,Z 300.748,A -85,B 0,C 180,E1 -8926.732,E2 -8926.732} C_VEL
LIN {X 0,Y 439.403,Z 300.748,A -85,B 0,C 180,E1 -8929.625,E2 -8929.625} C_VEL
LIN {X 0,Y 439.364,Z 300.754,A -85,B 0,C 180,E1 -8932.574,E2 -8932.574} C_VEL
LIN {X 0,Y 439.365,Z 300.751,A -85,B 0,C 180,E1 -8935.586,E2 -8935.586} C_VEL
LIN {X 0,Y 439.38,Z 300.753,A -85,B 0,C 180,E1 -8938.675,E2 -8938.675} C_VEL
LIN {X 0,Y 439.361,Z 300.754,A -85,B 0,C 180,E1 -8942.028,E2 -8942.028} C_VEL
LIN {X 0,Y 439.387,Z 300.748,A -85,B 0,C 180,E1 -8945.338,E2 -8945.338} C_VEL
LIN {X 0,Y 439.354,Z 300.759,A -85,B 0,C 180,E1 -8948.597,E2 -8948.597} C_VEL
LIN {X 0,Y 439.343,Z 300.755,A -85,B 0,C 180,E1 -8952.209,E2 -8952.209} C_VEL
LIN {X 0,Y 439.392,Z 300.751,A -85,B 0,C 180,E1 -8955.269,E2 -8955.269} C_VEL
LIN {X 0,Y 439.348,Z 300.761,A -85,B 0,C 180,E1 -8959.015,E2 -8959.015} C_VEL
LIN {X 0,Y 439.33,Z 300.757,A -85,B 0,C 180,E1 -8962.563,E2 -8962.563} C_VEL
LIN {X 0,Y 439.382,Z 300.752,A -85,B 0,C 180,E1 -8964.842,E2 -8964.842} C_VEL
LIN {X 0,Y 439.338,Z 300.754,A -85,B 0,C 180,E1 -8968.136,E2 -8968.136} C_VEL
LIN {X 0,Y 439.369,Z 300.757,A -85,B 0,C 180,E1 -8971.323,E2 -8971.323} C_VEL
LIN {X 0,Y 439.345,Z 300.753,A -85,B 0,C 180,E1 -8974.411,E2 -8974.411} C_VEL
LIN {X 0,Y 439.354,Z 300.758,A -85,B 0,C 180,E1 -8977.424,E2 -8977.424} C_VEL
LIN {X 0,Y 439.432,Z 300.742,A -85,B 0,C 180,E1 -8980.663,E2 -8980.663} C_VEL
LIN {X 0,Y 439.392,Z 300.75,A -85,B 0,C 180,E1 -8984.222,E2 -8984.222} C_VEL
LIN {X 0,Y 439.457,Z 300.74,A -85,B 0,C 180,E1 -8987.296,E2 -8987.296} C_VEL
LIN {X 0,Y 439.465,Z 300.739,A -85,B 0,C 180,E1 -8990.797,E2 -8990.797} C_VEL
LIN {X 0,Y 439.548,Z 300.73,A -85,B 0,C 180,E1 -8993.574,E2 -8993.574} C_VEL
LIN {X 0,Y 439.402,Z 300.746,A -85,B 0,C 180,E1 -8995.413,E2 -8995.413} C_VEL
LIN {X 0,Y 439.619,Z 300.726,A -85,B 0,C 180,E1 -8998.168,E2 -8998.168} C_VEL
LIN {X 0,Y 439.575,Z 300.726,A -85,B 0,C 180,E1 -9000.916,E2 -9000.916} C_VEL
LIN {X 0,Y 439.6,Z 300.725,A -85,B 0,C 180,E1 -9002.749,E2 -9002.749} C_VEL
LIN {X 0,Y 439.586,Z 300.73,A -85,B 0,C 180,E1 -9006.426,E2 -9006.426} C_VEL
LIN {X 0,Y 439.48,Z 300.738,A -85,B 0,C 180,E1 -9009.202,E2 -9009.202} C_VEL
LIN {X 0,Y 439.456,Z 300.745,A -85,B 0,C 180,E1 -9012.938,E2 -9012.938} C_VEL
LIN {X 0,Y 439.437,Z 300.744,A -85,B 0,C 180,E1 -9016.348,E2 -9016.348} C_VEL
LIN {X 0,Y 439.393,Z 300.748,A -85,B 0,C 180,E1 -9019.627,E2 -9019.627} C_VEL
LIN {X 0,Y 439.354,Z 300.754,A -85,B 0,C 180,E1 -9022.576,E2 -9022.576} C_VEL
LIN {X 0,Y 439.369,Z 300.753,A -85,B 0,C 180,E1 -9025.587,E2 -9025.587} C_VEL
LIN {X 0,Y 439.409,Z 300.747,A -85,B 0,C 180,E1 -9028.674,E2 -9028.674} C_VEL
LIN {X 0,Y 439.362,Z 300.752,A -85,B 0,C 180,E1 -9032.031,E2 -9032.031} C_VEL
LIN {X 0,Y 439.386,Z 300.755,A -85,B 0,C 180,E1 -9035.341,E2 -9035.341} C_VEL
LIN {X 0,Y 439.356,Z 300.752,A -85,B 0,C 180,E1 -9038.598,E2 -9038.598} C_VEL
LIN {X 0,Y 439.375,Z 300.753,A -85,B 0,C 180,E1 -9041.256,E2 -9041.256} C_VEL
LIN {X 0,Y 439.393,Z 300.747,A -85,B 0,C 180,E1 -9044.73,E2 -9044.73} C_VEL
LIN {X 0,Y 439.379,Z 300.757,A -85,B 0,C 180,E1 -9047.795,E2 -9047.795} C_VEL
LIN {X 0,Y 439.384,Z 300.753,A -85,B 0,C 180,E1 -9050.224,E2 -9050.224} C_VEL
LIN {X 0,Y 439.368,Z 300.754,A -85,B 0,C 180,E1 -9053.714,E2 -9053.714} C_VEL
LIN {X 0,Y 439.369,Z 300.75,A -85,B 0,C 180,E1 -9057.055,E2 -9057.055} C_VEL
LIN {X 0,Y 439.379,Z 300.757,A -85,B 0,C 180,E1 -9060.275,E2 -9060.275} C_VEL
LIN {X 0,Y 439.417,Z 300.748,A -85,B 0,C 180,E1 -9063.397,E2 -9063.397} C_VEL
LIN {X 0,Y 439.454,Z 300.942,A -85,B 0,C 180,E1 -9063.814,E2 -9063.814} C_VEL
LIN {X 0,Y 441.731,Z 313.243,A -85,B 0,C 180,E1 -9066.315,E2 -9066.315} C_VEL
LIN {X 0,Y 441.325,Z 323.554,A -85,B 0,C 180,E1 -9068.27,E2 -9068.27} C_VEL
LIN {X 0,Y 440.451,Z 341.633,A -85,B 0,C 180,E1 -9071.656,E2 -9071.656} C_VEL
LIN {X 0,Y 440.322,Z 343.776,A -85,B 0,C 180,E1 -9072.053,E2 -9072.053} C_VEL
LIN {X 0,Y 443.703,Z 365.93,A -85,B 0,C 180,E1 -9072.545,E2 -9072.545} C_VEL
LIN {X 0,Y 442.937,Z 452.371,A -85,B 0,C 180,E1 -9073.968,E2 -9073.968} C_VEL
LIN {X 0,Y 442.424,Z 466.305,A -85,B 0,C 180,E1 -9074.393,E2 -9074.393} C_VEL
LIN {X 0,Y 441.942,Z 478.786,A -85,B 0,C 180,E1 -9074.966,E2 -9074.966} C_VEL
LIN {X 0,Y 441.369,Z 490.713,A -85,B 0,C 180,E1 -9075.712,E2 -9075.712} C_VEL
LIN {X 0,Y 440.677,Z 502.908,A -85,B 0,C 180,E1 -9076.697,E2 -9076.697} C_VEL
LIN {X 0,Y 440.137,Z 513.49,A -85,B 0,C 180,E1 -9077.786,E2 -9077.786} C_VEL
LIN {X 0,Y 439.552,Z 522.575,A -85,B 0,C 180,E1 -9078.939,E2 -9078.939} C_VEL
LIN {X 0,Y 439.08,Z 531.442,A -85,B 0,C 180,E1 -9080.325,E2 -9080.325} C_VEL
LIN {X 0,Y 438.717,Z 538.525,A -85,B 0,C 180,E1 -9081.711,E2 -9081.711} C_VEL
LIN {X 0,Y 438.506,Z 544.18,A -85,B 0,C 180,E1 -9083.097,E2 -9083.097} C_VEL
LIN {X 0,Y 438.378,Z 548.624,A -85,B 0,C 180,E1 -9084.481,E2 -9084.481} C_VEL
LIN {X 0,Y 438.341,Z 550.968,A -85,B 0,C 180,E1 -9085.403,E2 -9085.403} C_VEL
LIN {X 0,Y 438.281,Z 552.88,A -85,B 0,C 180,E1 -9086.323,E2 -9086.323} C_VEL
LIN {X 0,Y 438.34,Z 554.349,A -85,B 0,C 180,E1 -9087.244,E2 -9087.244} C_VEL
LIN {X 0,Y 438.252,Z 556.022,A -85,B 0,C 180,E1 -9089.082,E2 -9089.082} C_VEL
LIN {X 0,Y 438.253,Z 556.278,A -85,B 0,C 180,E1 -9090.001,E2 -9090.001} C_VEL
LIN {X 0,Y 438.252,Z 556.124,A -85,B 0,C 180,E1 -9090.92,E2 -9090.92} C_VEL
LIN {X 0,Y 438.34,Z 554.59,A -85,B 0,C 180,E1 -9092.758,E2 -9092.758} C_VEL
LIN {X 0,Y 438.279,Z 553.232,A -85,B 0,C 180,E1 -9093.678,E2 -9093.678} C_VEL
LIN {X 0,Y 438.383,Z 550.371,A -85,B 0,C 180,E1 -9095.059,E2 -9095.059} C_VEL
LIN {X 0,Y 438.448,Z 546.486,A -85,B 0,C 180,E1 -9096.443,E2 -9096.443} C_VEL
LIN {X 0,Y 438.687,Z 541.483,A -85,B 0,C 180,E1 -9097.827,E2 -9097.827} C_VEL
LIN {X 0,Y 438.988,Z 535.209,A -85,B 0,C 180,E1 -9099.213,E2 -9099.213} C_VEL
LIN {X 0,Y 439.457,Z 527.37,A -85,B 0,C 180,E1 -9100.598,E2 -9100.598} C_VEL
LIN {X 0,Y 440.065,Z 519.391,A -85,B 0,C 180,E1 -9101.749,E2 -9101.749} C_VEL
LIN {X 0,Y 440.653,Z 509.677,A -85,B 0,C 180,E1 -9102.903,E2 -9102.903} C_VEL
LIN {X 0,Y 441.296,Z 498.896,A -85,B 0,C 180,E1 -9103.939,E2 -9103.939} C_VEL
LIN {X 0,Y 441.969,Z 488.393,A -85,B 0,C 180,E1 -9104.74,E2 -9104.74} C_VEL
LIN {X 0,Y 442.673,Z 475.768,A -85,B 0,C 180,E1 -9105.482,E2 -9105.482} C_VEL
LIN {X 0,Y 443.239,Z 463.174,A -85,B 0,C 180,E1 -9106.022,E2 -9106.022} C_VEL
LIN {X 0,Y 443.626,Z 449.869,A -85,B 0,C 180,E1 -9106.391,E2 -9106.391} C_VEL
LIN {X 0,Y 444.429,Z 365.491,A -85,B 0,C 180,E1 -9107.789,E2 -9107.789} C_VEL
LIN {X 0,Y 440.658,Z 343.427,A -85,B 0,C 180,E1 -9108.367,E2 -9108.367} C_VEL
LIN {X 0,Y 441.757,Z 324.538,A -85,B 0,C 180,E1 -9111.955,E2 -9111.955} C_VEL
LIN {X 0,Y 442.258,Z 315.718,A -85,B 0,C 180,E1 -9113.657,E2 -9113.657} C_VEL
LIN {X 0,Y 440.751,Z 306.911,A -85,B 0,C 180,E1 -9115.502,E2 -9115.502} C_VEL
LIN {X 0,Y 439.426,Z 300.752,A -85,B 0,C 180,E1 -9116.861,E2 -9116.861} C_VEL
LIN {X 0,Y 439.384,Z 300.758,A -85,B 0,C 180,E1 -9119.726,E2 -9119.726} C_VEL
LIN {X 0,Y 439.375,Z 300.755,A -85,B 0,C 180,E1 -9122.946,E2 -9122.946} C_VEL
LIN {X 0,Y 439.374,Z 300.758,A -85,B 0,C 180,E1 -9126.288,E2 -9126.288} C_VEL
LIN {X 0,Y 439.378,Z 300.754,A -85,B 0,C 180,E1 -9129.845,E2 -9129.845} C_VEL
LIN {X 0,Y 439.372,Z 300.755,A -85,B 0,C 180,E1 -9132.625,E2 -9132.625} C_VEL
LIN {X 0,Y 439.4,Z 300.748,A -85,B 0,C 180,E1 -9135.271,E2 -9135.271} C_VEL
LIN {X 0,Y 439.383,Z 300.753,A -85,B 0,C 180,E1 -9138.744,E2 -9138.744} C_VEL
LIN {X 0,Y 439.366,Z 300.748,A -85,B 0,C 180,E1 -9141.609,E2 -9141.609} C_VEL
LIN {X 0,Y 439.399,Z 300.751,A -85,B 0,C 180,E1 -9144.844,E2 -9144.844} C_VEL
LIN {X 0,Y 439.373,Z 300.748,A -85,B 0,C 180,E1 -9148.14,E2 -9148.14} C_VEL
LIN {X 0,Y 439.41,Z 300.745,A -85,B 0,C 180,E1 -9151.604,E2 -9151.604} C_VEL
LIN {X 0,Y 439.378,Z 300.75,A -85,B 0,C 180,E1 -9154.413,E2 -9154.413} C_VEL
LIN {X 0,Y 439.364,Z 300.756,A -85,B 0,C 180,E1 -9157.425,E2 -9157.425} C_VEL
LIN {X 0,Y 439.442,Z 300.742,A -85,B 0,C 180,E1 -9160.663,E2 -9160.663} C_VEL
LIN {X 0,Y 439.463,Z 300.738,A -85,B 0,C 180,E1 -9164.225,E2 -9164.225} C_VEL
LIN {X 0,Y 439.484,Z 300.737,A -85,B 0,C 180,E1 -9168.001,E2 -9168.001} C_VEL
LIN {X 0,Y 439.505,Z 300.734,A -85,B 0,C 180,E1 -9171.726,E2 -9171.726} C_VEL
LIN {X 0,Y 439.615,Z 300.718,A -85,B 0,C 180,E1 -9174.496,E2 -9174.496} C_VEL
LIN {X 0,Y 439.631,Z 300.722,A -85,B 0,C 180,E1 -9178.168,E2 -9178.168} C_VEL
LIN {X 0,Y 439.759,Z 300.703,A -85,B 0,C 180,E1 -9180,E2 -9180} C_VEL
LIN {X 0,Y 439.632,Z 300.718,A -85,B 0,C 180,E1 -9182.749,E2 -9182.749} C_VEL
LIN {X 0,Y 439.592,Z 300.729,A -85,B 0,C 180,E1 -9186.426,E2 -9186.426} C_VEL
LIN {X 0,Y 439.497,Z 300.731,A -85,B 0,C 180,E1 -9189.202,E2 -9189.202} C_VEL
LIN {X 0,Y 439.467,Z 300.738,A -85,B 0,C 180,E1 -9192.938,E2 -9192.938} C_VEL
LIN {X 0,Y 439.448,Z 300.745,A -85,B 0,C 180,E1 -9196.348,E2 -9196.348} C_VEL
LIN {X 0,Y 439.404,Z 300.747,A -85,B 0,C 180,E1 -9199.627,E2 -9199.627} C_VEL
LIN {X 0,Y 439.366,Z 300.751,A -85,B 0,C 180,E1 -9202.576,E2 -9202.576} C_VEL
LIN {X 0,Y 439.382,Z 300.749,A -85,B 0,C 180,E1 -9205.587,E2 -9205.587} C_VEL
LIN {X 0,Y 439.402,Z 300.746,A -85,B 0,C 180,E1 -9208.675,E2 -9208.675} C_VEL
LIN {X 0,Y 439.371,Z 300.75,A -85,B 0,C 180,E1 -9212.03,E2 -9212.03} C_VEL
LIN {X 0,Y 439.394,Z 300.752,A -85,B 0,C 180,E1 -9215.34,E2 -9215.34} C_VEL
LIN {X 0,Y 439.372,Z 300.752,A -85,B 0,C 180,E1 -9218.597,E2 -9218.597} C_VEL
LIN {X 0,Y 439.384,Z 300.753,A -85,B 0,C 180,E1 -9221.256,E2 -9221.256} C_VEL
LIN {X 0,Y 439.402,Z 300.749,A -85,B 0,C 180,E1 -9224.73,E2 -9224.73} C_VEL
LIN {X 0,Y 439.362,Z 300.759,A -85,B 0,C 180,E1 -9227.791,E2 -9227.791} C_VEL
LIN {X 0,Y 439.365,Z 300.758,A -85,B 0,C 180,E1 -9231.403,E2 -9231.403} C_VEL
LIN {X 0,Y 439.398,Z 300.753,A -85,B 0,C 180,E1 -9234.844,E2 -9234.844} C_VEL
LIN {X 0,Y 439.423,Z 300.945,A -85,B 0,C 180,E1 -9236.452,E2 -9236.452} C_VEL
LIN {X 0,Y 441.087,Z 309.045,A -85,B 0,C 180,E1 -9238.277,E2 -9238.277} C_VEL
LIN {X 0,Y 441.07,Z 316.664,A -85,B 0,C 180,E1 -9239.872,E2 -9239.872} C_VEL
LIN {X 0,Y 440.912,Z 320.796,A -85,B 0,C 180,E1 -9240.714,E2 -9240.714} C_VEL
LIN {X 0,Y 444.717,Z 339.021,A -85,B 0,C 180,E1 -9241.209,E2 -9241.209} C_VEL
LIN {X 0,Y 443.714,Z 428.08,A -85,B 0,C 180,E1 -9242.687,E2 -9242.687} C_VEL
LIN {X 0,Y 443.403,Z 440.242,A -85,B 0,C 180,E1 -9243.049,E2 -9243.049} C_VEL
LIN {X 0,Y 442.92,Z 451.958,A -85,B 0,C 180,E1 -9243.558,E2 -9243.558} C_VEL
LIN {X 0,Y 442.43,Z 463.304,A -85,B 0,C 180,E1 -9244.224,E2 -9244.224} C_VEL
LIN {X 0,Y 441.804,Z 474.419,A -85,B 0,C 180,E1 -9245.058,E2 -9245.058} C_VEL
LIN {X 0,Y 441.129,Z 484.703,A -85,B 0,C 180,E1 -9246.029,E2 -9246.029} C_VEL
LIN {X 0,Y 440.422,Z 494.934,A -85,B 0,C 180,E1 -9247.234,E2 -9247.234} C_VEL
LIN {X 0,Y 439.88,Z 503.253,A -85,B 0,C 180,E1 -9248.44,E2 -9248.44} C_VEL
LIN {X 0,Y 439.625,Z 507.372,A -85,B 0,C 180,E1 -9249.136,E2 -9249.136} C_VEL
LIN {X 0,Y 438.825,Z 510.822,A -85,B 0,C 180,E1 -9249.751,E2 -9249.751} C_VEL
LIN {X 0,Y 435.661,Z 515.98,A -85,B 0,C 180,E1 -9250.781,E2 -9250.781} C_VEL
LIN {X 0,Y 432.455,Z 520.434,A -85,B 0,C 180,E1 -9251.876,E2 -9251.876} C_VEL
LIN {X 0,Y 431.605,Z 522.781,A -85,B 0,C 180,E1 -9252.589,E2 -9252.589} C_VEL
LIN {X 0,Y 431.426,Z 526.452,A -85,B 0,C 180,E1 -9253.972,E2 -9253.972} C_VEL
LIN {X 0,Y 431.306,Z 528.342,A -85,B 0,C 180,E1 -9254.887,E2 -9254.887} C_VEL
LIN {X 0,Y 431.176,Z 529.909,A -85,B 0,C 180,E1 -9255.848,E2 -9255.848} C_VEL
LIN {X 0,Y 431.136,Z 531.005,A -85,B 0,C 180,E1 -9256.807,E2 -9256.807} C_VEL
LIN {X 0,Y 431.203,Z 531.768,A -85,B 0,C 180,E1 -9257.938,E2 -9257.938} C_VEL
LIN {X 0,Y 431.119,Z 531.851,A -85,B 0,C 180,E1 -9259.669,E2 -9259.669} C_VEL
LIN {X 0,Y 431.155,Z 530.338,A -85,B 0,C 180,E1 -9261.563,E2 -9261.563} C_VEL
LIN {X 0,Y 431.238,Z 528.989,A -85,B 0,C 180,E1 -9262.508,E2 -9262.508} C_VEL
LIN {X 0,Y 431.358,Z 526.754,A -85,B 0,C 180,E1 -9263.65,E2 -9263.65} C_VEL
LIN {X 0,Y 431.476,Z 522.276,A -85,B 0,C 180,E1 -9265.328,E2 -9265.328} C_VEL
LIN {X 0,Y 431.763,Z 517.28,A -85,B 0,C 180,E1 -9266.733,E2 -9266.733} C_VEL
LIN {X 0,Y 432.014,Z 511.029,A -85,B 0,C 180,E1 -9268.135,E2 -9268.135} C_VEL
LIN {X 0,Y 432.592,Z 503.182,A -85,B 0,C 180,E1 -9269.534,E2 -9269.534} C_VEL
LIN {X 0,Y 432.978,Z 495.232,A -85,B 0,C 180,E1 -9270.697,E2 -9270.697} C_VEL
LIN {X 0,Y 433.464,Z 486.6,A -85,B 0,C 180,E1 -9271.741,E2 -9271.741} C_VEL
LIN {X 0,Y 434.256,Z 475.995,A -85,B 0,C 180,E1 -9272.782,E2 -9272.782} C_VEL
LIN {X 0,Y 434.786,Z 465.799,A -85,B 0,C 180,E1 -9273.59,E2 -9273.59} C_VEL
LIN {X 0,Y 435.289,Z 453.689,A -85,B 0,C 180,E1 -9274.34,E2 -9274.34} C_VEL
LIN {X 0,Y 435.703,Z 440.241,A -85,B 0,C 180,E1 -9274.944,E2 -9274.944} C_VEL
LIN {X 0,Y 436.01,Z 427.631,A -85,B 0,C 180,E1 -9275.317,E2 -9275.317} C_VEL
LIN {X 0,Y 436.946,Z 339.287,A -85,B 0,C 180,E1 -9276.783,E2 -9276.783} C_VEL
LIN {X 0,Y 433.518,Z 320.842,A -85,B 0,C 180,E1 -9277.246,E2 -9277.246} C_VEL
LIN {X 0,Y 434.009,Z 310.978,A -85,B 0,C 180,E1 -9279.318,E2 -9279.318} C_VEL
LIN {X 0,Y 432.445,Z 301.622,A -85,B 0,C 180,E1 -9281.423,E2 -9281.423} C_VEL
LIN {X 0,Y 432.361,Z 301.631,A -85,B 0,C 180,E1 -9284.111,E2 -9284.111} C_VEL
LIN {X 0,Y 432.332,Z 301.627,A -85,B 0,C 180,E1 -9287.013,E2 -9287.013} C_VEL
LIN {X 0,Y 432.339,Z 301.632,A -85,B 0,C 180,E1 -9289.959,E2 -9289.959} C_VEL
LIN {X 0,Y 432.312,Z 301.63,A -85,B 0,C 180,E1 -9292.964,E2 -9292.964} C_VEL
LIN {X 0,Y 432.317,Z 301.633,A -85,B 0,C 180,E1 -9296.034,E2 -9296.034} C_VEL
LIN {X 0,Y 432.32,Z 301.629,A -85,B 0,C 180,E1 -9299.188,E2 -9299.188} C_VEL
LIN {X 0,Y 432.318,Z 301.636,A -85,B 0,C 180,E1 -9302.442,E2 -9302.442} C_VEL
LIN {X 0,Y 432.332,Z 301.627,A -85,B 0,C 180,E1 -9305.817,E2 -9305.817} C_VEL
LIN {X 0,Y 432.297,Z 301.632,A -85,B 0,C 180,E1 -9309.347,E2 -9309.347} C_VEL
LIN {X 0,Y 432.299,Z 301.631,A -85,B 0,C 180,E1 -9311.8,E2 -9311.8} C_VEL
LIN {X 0,Y 432.329,Z 301.629,A -85,B 0,C 180,E1 -9314.346,E2 -9314.346} C_VEL
LIN {X 0,Y 432.295,Z 301.639,A -85,B 0,C 180,E1 -9317.018,E2 -9317.018} C_VEL
LIN {X 0,Y 432.283,Z 301.633,A -85,B 0,C 180,E1 -9319.827,E2 -9319.827} C_VEL
LIN {X 0,Y 432.291,Z 301.638,A -85,B 0,C 180,E1 -9323.02,E2 -9323.02} C_VEL
LIN {X 0,Y 432.324,Z 301.628,A -85,B 0,C 180,E1 -9326.002,E2 -9326.002} C_VEL
LIN {X 0,Y 432.323,Z 301.634,A -85,B 0,C 180,E1 -9329.493,E2 -9329.493} C_VEL
LIN {X 0,Y 432.304,Z 301.633,A -85,B 0,C 180,E1 -9331.871,E2 -9331.871} C_VEL
LIN {X 0,Y 432.339,Z 301.634,A -85,B 0,C 180,E1 -9335.547,E2 -9335.547} C_VEL
LIN {X 0,Y 432.339,Z 301.627,A -85,B 0,C 180,E1 -9339.045,E2 -9339.045} C_VEL
LIN {X 0,Y 432.316,Z 301.634,A -85,B 0,C 180,E1 -9342.008,E2 -9342.008} C_VEL
LIN {X 0,Y 432.317,Z 301.629,A -85,B 0,C 180,E1 -9344.923,E2 -9344.923} C_VEL
LIN {X 0,Y 432.44,Z 301.62,A -85,B 0,C 180,E1 -9347.803,E2 -9347.803} C_VEL
LIN {X 0,Y 432.437,Z 301.616,A -85,B 0,C 180,E1 -9351.589,E2 -9351.589} C_VEL
LIN {X 0,Y 432.54,Z 301.606,A -85,B 0,C 180,E1 -9354.405,E2 -9354.405} C_VEL
LIN {X 0,Y 432.589,Z 301.601,A -85,B 0,C 180,E1 -9358.138,E2 -9358.138} C_VEL
LIN {X 0,Y 432.536,Z 301.603,A -85,B 0,C 180,E1 -9360.931,E2 -9360.931} C_VEL
LIN {X 0,Y 432.553,Z 301.603,A -85,B 0,C 180,E1 -9362.794,E2 -9362.794} C_VEL
LIN {X 0,Y 432.575,Z 301.597,A -85,B 0,C 180,E1 -9365.594,E2 -9365.594} C_VEL
LIN {X 0,Y 432.453,Z 301.617,A -85,B 0,C 180,E1 -9368.41,E2 -9368.41} C_VEL
LIN {X 0,Y 432.449,Z 301.614,A -85,B 0,C 180,E1 -9372.197,E2 -9372.197} C_VEL
LIN {X 0,Y 432.421,Z 301.616,A -85,B 0,C 180,E1 -9376.039,E2 -9376.039} C_VEL
LIN {X 0,Y 432.378,Z 301.623,A -85,B 0,C 180,E1 -9379.485,E2 -9379.485} C_VEL
LIN {X 0,Y 432.308,Z 301.637,A -85,B 0,C 180,E1 -9382.965,E2 -9382.965} C_VEL
LIN {X 0,Y 432.329,Z 301.634,A -85,B 0,C 180,E1 -9385.003,E2 -9385.003} C_VEL
LIN {X 0,Y 432.372,Z 301.622,A -85,B 0,C 180,E1 -9388.124,E2 -9388.124} C_VEL
LIN {X 0,Y 432.313,Z 301.638,A -85,B 0,C 180,E1 -9391.347,E2 -9391.347} C_VEL
LIN {X 0,Y 432.332,Z 301.627,A -85,B 0,C 180,E1 -9394.678,E2 -9394.678} C_VEL
LIN {X 0,Y 432.323,Z 301.629,A -85,B 0,C 180,E1 -9398.151,E2 -9398.151} C_VEL
LIN {X 0,Y 432.318,Z 301.636,A -85,B 0,C 180,E1 -9401.601,E2 -9401.601} C_VEL
LIN {X 0,Y 432.328,Z 301.629,A -85,B 0,C 180,E1 -9404.348,E2 -9404.348} C_VEL
LIN {X 0,Y 432.311,Z 301.63,A -85,B 0,C 180,E1 -9407.017,E2 -9407.017} C_VEL
LIN {X 0,Y 432.327,Z 301.634,A -85,B 0,C 180,E1 -9409.822,E2 -9409.822} C_VEL
LIN {X 0,Y 432.3,Z 301.631,A -85,B 0,C 180,E1 -9413.023,E2 -9413.023} C_VEL
LIN {X 0,Y 432.356,Z 301.63,A -85,B 0,C 180,E1 -9415.997,E2 -9415.997} C_VEL
LIN {X 0,Y 432.345,Z 301.626,A -85,B 0,C 180,E1 -9419.491,E2 -9419.491} C_VEL
LIN {X 0,Y 432.383,Z 301.626,A -85,B 0,C 180,E1 -9422.929,E2 -9422.929} C_VEL
LIN {X 0,Y 432.417,Z 301.731,A -85,B 0,C 180,E1 -9423.602,E2 -9423.602} C_VEL
LIN {X 0,Y 434.704,Z 314.102,A -85,B 0,C 180,E1 -9426.161,E2 -9426.161} C_VEL
LIN {X 0,Y 434.579,Z 320.008,A -85,B 0,C 180,E1 -9427.307,E2 -9427.307} C_VEL
LIN {X 0,Y 433.709,Z 337.265,A -85,B 0,C 180,E1 -9430.599,E2 -9430.599} C_VEL
LIN {X 0,Y 433.382,Z 343.644,A -85,B 0,C 180,E1 -9431.799,E2 -9431.799} C_VEL
LIN {X 0,Y 436.861,Z 367.849,A -85,B 0,C 180,E1 -9432.335,E2 -9432.335} C_VEL
LIN {X 0,Y 436.06,Z 451.972,A -85,B 0,C 180,E1 -9433.739,E2 -9433.739} C_VEL
LIN {X 0,Y 435.551,Z 465.205,A -85,B 0,C 180,E1 -9434.14,E2 -9434.14} C_VEL
LIN {X 0,Y 435.081,Z 477.953,A -85,B 0,C 180,E1 -9434.723,E2 -9434.723} C_VEL
LIN {X 0,Y 434.43,Z 490.053,A -85,B 0,C 180,E1 -9435.479,E2 -9435.479} C_VEL
LIN {X 0,Y 433.729,Z 502.167,A -85,B 0,C 180,E1 -9436.464,E2 -9436.464} C_VEL
LIN {X 0,Y 433.138,Z 512.001,A -85,B 0,C 180,E1 -9437.467,E2 -9437.467} C_VEL
LIN {X 0,Y 432.671,Z 520.498,A -85,B 0,C 180,E1 -9438.523,E2 -9438.523} C_VEL
LIN {X 0,Y 432.106,Z 529.692,A -85,B 0,C 180,E1 -9439.931,E2 -9439.931} C_VEL
LIN {X 0,Y 431.732,Z 537.092,A -85,B 0,C 180,E1 -9441.34,E2 -9441.34} C_VEL
LIN {X 0,Y 431.423,Z 543.873,A -85,B 0,C 180,E1 -9442.983,E2 -9442.983} C_VEL
LIN {X 0,Y 431.281,Z 548.343,A -85,B 0,C 180,E1 -9444.39,E2 -9444.39} C_VEL
LIN {X 0,Y 431.27,Z 550.701,A -85,B 0,C 180,E1 -9445.327,E2 -9445.327} C_VEL
LIN {X 0,Y 431.187,Z 552.623,A -85,B 0,C 180,E1 -9446.263,E2 -9446.263} C_VEL
LIN {X 0,Y 431.236,Z 554.114,A -85,B 0,C 180,E1 -9447.198,E2 -9447.198} C_VEL
LIN {X 0,Y 431.202,Z 555.156,A -85,B 0,C 180,E1 -9448.133,E2 -9448.133} C_VEL
LIN {X 0,Y 431.167,Z 556.074,A -85,B 0,C 180,E1 -9450.001,E2 -9450.001} C_VEL
LIN {X 0,Y 431.168,Z 555.94,A -85,B 0,C 180,E1 -9450.935,E2 -9450.935} C_VEL
LIN {X 0,Y 431.202,Z 555.377,A -85,B 0,C 180,E1 -9451.869,E2 -9451.869} C_VEL
LIN {X 0,Y 431.235,Z 554.426,A -85,B 0,C 180,E1 -9452.803,E2 -9452.803} C_VEL
LIN {X 0,Y 431.186,Z 553.08,A -85,B 0,C 180,E1 -9453.739,E2 -9453.739} C_VEL
LIN {X 0,Y 431.294,Z 550.241,A -85,B 0,C 180,E1 -9455.143,E2 -9455.143} C_VEL
LIN {X 0,Y 431.377,Z 546.381,A -85,B 0,C 180,E1 -9456.549,E2 -9456.549} C_VEL
LIN {X 0,Y 431.611,Z 541.405,A -85,B 0,C 180,E1 -9457.956,E2 -9457.956} C_VEL
LIN {X 0,Y 431.975,Z 535.164,A -85,B 0,C 180,E1 -9459.364,E2 -9459.364} C_VEL
LIN {X 0,Y 432.46,Z 527.379,A -85,B 0,C 180,E1 -9460.772,E2 -9460.772} C_VEL
LIN {X 0,Y 433.113,Z 519.445,A -85,B 0,C 180,E1 -9461.941,E2 -9461.941} C_VEL
LIN {X 0,Y 433.736,Z 509.785,A -85,B 0,C 180,E1 -9463.112,E2 -9463.112} C_VEL
LIN {X 0,Y 434.416,Z 499.077,A -85,B 0,C 180,E1 -9464.164,E2 -9464.164} C_VEL
LIN {X 0,Y 435.109,Z 488.699,A -85,B 0,C 180,E1 -9464.978,E2 -9464.978} C_VEL
LIN {X 0,Y 435.86,Z 476.245,A -85,B 0,C 180,E1 -9465.73,E2 -9465.73} C_VEL
LIN {X 0,Y 436.493,Z 463.136,A -85,B 0,C 180,E1 -9466.306,E2 -9466.306} C_VEL
LIN {X 0,Y 436.892,Z 450.005,A -85,B 0,C 180,E1 -9466.681,E2 -9466.681} C_VEL
LIN {X 0,Y 437.716,Z 366.131,A -85,B 0,C 180,E1 -9468.095,E2 -9468.095} C_VEL
LIN {X 0,Y 433.797,Z 343.232,A -85,B 0,C 180,E1 -9468.706,E2 -9468.706} C_VEL
LIN {X 0,Y 434.918,Z 324.558,A -85,B 0,C 180,E1 -9472.318,E2 -9472.318} C_VEL
LIN {X 0,Y 435.349,Z 317.002,A -85,B 0,C 180,E1 -9473.803,E2 -9473.803} C_VEL
LIN {X 0,Y 433.537,Z 306.952,A -85,B 0,C 180,E1 -9475.957,E2 -9475.957} C_VEL
LIN {X 0,Y 432.403,Z 301.628,A -85,B 0,C 180,E1 -9477.137,E2 -9477.137} C_VEL
LIN {X 0,Y 432.35,Z 301.636,A -85,B 0,C 180,E1 -9480.511,E2 -9480.511} C_VEL
LIN {X 0,Y 432.362,Z 301.633,A -85,B 0,C 180,E1 -9484.004,E2 -9484.004} C_VEL
LIN {X 0,Y 432.322,Z 301.632,A -85,B 0,C 180,E1 -9487.197,E2 -9487.197} C_VEL
LIN {X 0,Y 432.313,Z 301.634,A -85,B 0,C 180,E1 -9490.562,E2 -9490.562} C_VEL
LIN {X 0,Y 432.316,Z 301.631,A -85,B 0,C 180,E1 -9493.062,E2 -9493.062} C_VEL
LIN {X 0,Y 432.335,Z 301.629,A -85,B 0,C 180,E1 -9495.665,E2 -9495.665} C_VEL
LIN {X 0,Y 432.326,Z 301.634,A -85,B 0,C 180,E1 -9498.399,E2 -9498.399} C_VEL
LIN {X 0,Y 432.331,Z 301.625,A -85,B 0,C 180,E1 -9501.849,E2 -9501.849} C_VEL
LIN {X 0,Y 432.34,Z 301.628,A -85,B 0,C 180,E1 -9505.323,E2 -9505.323} C_VEL
LIN {X 0,Y 432.322,Z 301.63,A -85,B 0,C 180,E1 -9508.654,E2 -9508.654} C_VEL
LIN {X 0,Y 432.348,Z 301.624,A -85,B 0,C 180,E1 -9511.874,E2 -9511.874} C_VEL
LIN {X 0,Y 432.378,Z 301.624,A -85,B 0,C 180,E1 -9515.539,E2 -9515.539} C_VEL
LIN {X 0,Y 432.351,Z 301.628,A -85,B 0,C 180,E1 -9519.046,E2 -9519.046} C_VEL
LIN {X 0,Y 432.362,Z 301.623,A -85,B 0,C 180,E1 -9522.011,E2 -9522.011} C_VEL
LIN {X 0,Y 432.395,Z 301.619,A -85,B 0,C 180,E1 -9524.927,E2 -9524.927} C_VEL
LIN {X 0,Y 432.46,Z 301.613,A -85,B 0,C 180,E1 -9527.804,E2 -9527.804} C_VEL
LIN {X 0,Y 432.465,Z 301.611,A -85,B 0,C 180,E1 -9531.59,E2 -9531.59} C_VEL
LIN {X 0,Y 432.591,Z 301.594,A -85,B 0,C 180,E1 -9534.406,E2 -9534.406} C_VEL
LIN {X 0,Y 432.601,Z 301.598,A -85,B 0,C 180,E1 -9538.138,E2 -9538.138} C_VEL
LIN {X 0,Y 432.729,Z 301.579,A -85,B 0,C 180,E1 -9540,E2 -9540} C_VEL
LIN {X 0,Y 432.584,Z 301.596,A -85,B 0,C 180,E1 -9542.794,E2 -9542.794} C_VEL
LIN {X 0,Y 432.586,Z 301.592,A -85,B 0,C 180,E1 -9545.594,E2 -9545.594} C_VEL
LIN {X 0,Y 432.465,Z 301.613,A -85,B 0,C 180,E1 -9548.41,E2 -9548.41} C_VEL
LIN {X 0,Y 432.461,Z 301.615,A -85,B 0,C 180,E1 -9552.197,E2 -9552.197} C_VEL
LIN {X 0,Y 432.432,Z 301.616,A -85,B 0,C 180,E1 -9556.039,E2 -9556.039} C_VEL
LIN {X 0,Y 432.388,Z 301.621,A -85,B 0,C 180,E1 -9559.485,E2 -9559.485} C_VEL
LIN {X 0,Y 432.319,Z 301.634,A -85,B 0,C 180,E1 -9562.965,E2 -9562.965} C_VEL
LIN {X 0,Y 432.341,Z 301.628,A -85,B 0,C 180,E1 -9565.002,E2 -9565.002} C_VEL
LIN {X 0,Y 432.349,Z 301.622,A -85,B 0,C 180,E1 -9568.126,E2 -9568.126} C_VEL
LIN {X 0,Y 432.323,Z 301.632,A -85,B 0,C 180,E1 -9571.346,E2 -9571.346} C_VEL
LIN {X 0,Y 432.339,Z 301.625,A -85,B 0,C 180,E1 -9574.678,E2 -9574.678} C_VEL
LIN {X 0,Y 432.335,Z 301.63,A -85,B 0,C 180,E1 -9578.151,E2 -9578.151} C_VEL
LIN {X 0,Y 432.327,Z 301.634,A -85,B 0,C 180,E1 -9581.601,E2 -9581.601} C_VEL
LIN {X 0,Y 432.337,Z 301.631,A -85,B 0,C 180,E1 -9584.347,E2 -9584.347} C_VEL
LIN {X 0,Y 432.31,Z 301.633,A -85,B 0,C 180,E1 -9587.018,E2 -9587.018} C_VEL
LIN {X 0,Y 432.294,Z 301.635,A -85,B 0,C 180,E1 -9589.828,E2 -9589.828} C_VEL
LIN {X 0,Y 432.307,Z 301.636,A -85,B 0,C 180,E1 -9593.022,E2 -9593.022} C_VEL
LIN {X 0,Y 432.372,Z 301.772,A -85,B 0,C 180,E1 -9596.159,E2 -9596.159} C_VEL
LIN {X 0,Y 434.235,Z 310.961,A -85,B 0,C 180,E1 -9598.264,E2 -9598.264} C_VEL
LIN {X 0,Y 434.04,Z 321.003,A -85,B 0,C 180,E1 -9600.37,E2 -9600.37} C_VEL
LIN {X 0,Y 438.028,Z 339.867,A -85,B 0,C 180,E1 -9600.899,E2 -9600.899} C_VEL
LIN {X 0,Y 437.003,Z 428.389,A -85,B 0,C 180,E1 -9602.395,E2 -9602.395} C_VEL
LIN {X 0,Y 436.661,Z 440.505,A -85,B 0,C 180,E1 -9602.761,E2 -9602.761} C_VEL
LIN {X 0,Y 436.13,Z 452.79,A -85,B 0,C 180,E1 -9603.308,E2 -9603.308} C_VEL
LIN {X 0,Y 435.594,Z 464.919,A -85,B 0,C 180,E1 -9604.046,E2 -9604.046} C_VEL
LIN {X 0,Y 434.892,Z 476.219,A -85,B 0,C 180,E1 -9604.941,E2 -9604.941} C_VEL
LIN {X 0,Y 434.103,Z 486.848,A -85,B 0,C 180,E1 -9605.998,E2 -9605.998} C_VEL
LIN {X 0,Y 433.386,Z 497.065,A -85,B 0,C 180,E1 -9607.267,E2 -9607.267} C_VEL
LIN {X 0,Y 432.784,Z 505.456,A -85,B 0,C 180,E1 -9608.569,E2 -9608.569} C_VEL
LIN {X 0,Y 432.202,Z 513.085,A -85,B 0,C 180,E1 -9610.032,E2 -9610.032} C_VEL
LIN {X 0,Y 431.838,Z 519.15,A -85,B 0,C 180,E1 -9611.496,E2 -9611.496} C_VEL
LIN {X 0,Y 431.605,Z 522.781,A -85,B 0,C 180,E1 -9612.589,E2 -9612.589} C_VEL
LIN {X 0,Y 430.786,Z 524.906,A -85,B 0,C 180,E1 -9613.316,E2 -9613.316} C_VEL
LIN {X 0,Y 427.721,Z 527.845,A -85,B 0,C 180,E1 -9614.514,E2 -9614.514} C_VEL
LIN {X 0,Y 425.208,Z 529.665,A -85,B 0,C 180,E1 -9615.499,E2 -9615.499} C_VEL
LIN {X 0,Y 424.147,Z 530.719,A -85,B 0,C 180,E1 -9616.272,E2 -9616.272} C_VEL
LIN {X 0,Y 424.066,Z 531.015,A -85,B 0,C 180,E1 -9616.534,E2 -9616.534} C_VEL
LIN {X 0,Y 424.109,Z 531.965,A -85,B 0,C 180,E1 -9617.88,E2 -9617.88} C_VEL
LIN {X 0,Y 424.036,Z 532.085,A -85,B 0,C 180,E1 -9619.495,E2 -9619.495} C_VEL
LIN {X 0,Y 424,Z 531.618,A -85,B 0,C 180,E1 -9620.458,E2 -9620.458} C_VEL
LIN {X 0,Y 424.063,Z 530.714,A -85,B 0,C 180,E1 -9621.421,E2 -9621.421} C_VEL
LIN {X 0,Y 424.126,Z 529.416,A -85,B 0,C 180,E1 -9622.382,E2 -9622.382} C_VEL
LIN {X 0,Y 424.268,Z 526.995,A -85,B 0,C 180,E1 -9623.673,E2 -9623.673} C_VEL
LIN {X 0,Y 424.392,Z 522.915,A -85,B 0,C 180,E1 -9625.25,E2 -9625.25} C_VEL
LIN {X 0,Y 424.667,Z 518.038,A -85,B 0,C 180,E1 -9626.679,E2 -9626.679} C_VEL
LIN {X 0,Y 424.919,Z 511.92,A -85,B 0,C 180,E1 -9628.104,E2 -9628.104} C_VEL
LIN {X 0,Y 425.521,Z 504.288,A -85,B 0,C 180,E1 -9629.526,E2 -9629.526} C_VEL
LIN {X 0,Y 426.027,Z 494.749,A -85,B 0,C 180,E1 -9630.945,E2 -9630.945} C_VEL
LIN {X 0,Y 426.623,Z 485.96,A -85,B 0,C 180,E1 -9632.005,E2 -9632.005} C_VEL
LIN {X 0,Y 427.374,Z 475.19,A -85,B 0,C 180,E1 -9633.063,E2 -9633.063} C_VEL
LIN {X 0,Y 428.018,Z 462.96,A -85,B 0,C 180,E1 -9634.001,E2 -9634.001} C_VEL
LIN {X 0,Y 428.474,Z 451.039,A -85,B 0,C 180,E1 -9634.703,E2 -9634.703} C_VEL
LIN {X 0,Y 428.863,Z 438.809,A -85,B 0,C 180,E1 -9635.229,E2 -9635.229} C_VEL
LIN {X 0,Y 429.214,Z 426.152,A -85,B 0,C 180,E1 -9635.578,E2 -9635.578} C_VEL
LIN {X 0,Y 430.198,Z 340.899,A -85,B 0,C 180,E1 -9637.008,E2 -9637.008} C_VEL
LIN {X 0,Y 426.593,Z 321.014,A -85,B 0,C 180,E1 -9637.513,E2 -9637.513} C_VEL
LIN {X 0,Y 426.998,Z 311.823,A -85,B 0,C 180,E1 -9639.473,E2 -9639.473} C_VEL
LIN {X 0,Y 425.403,Z 302.498,A -85,B 0,C 180,E1 -9641.615,E2 -9641.615} C_VEL
LIN {X 0,Y 425.33,Z 302.505,A -85,B 0,C 180,E1 -9644.35,E2 -9644.35} C_VEL
LIN {X 0,Y 425.298,Z 302.504,A -85,B 0,C 180,E1 -9647.303,E2 -9647.303} C_VEL
LIN {X 0,Y 425.296,Z 302.509,A -85,B 0,C 180,E1 -9650.304,E2 -9650.304} C_VEL
LIN {X 0,Y 425.271,Z 302.507,A -85,B 0,C 180,E1 -9653.366,E2 -9653.366} C_VEL
LIN {X 0,Y 425.286,Z 302.51,A -85,B 0,C 180,E1 -9656.498,E2 -9656.498} C_VEL
LIN {X 0,Y 425.277,Z 302.506,A -85,B 0,C 180,E1 -9659.719,E2 -9659.719} C_VEL
LIN {X 0,Y 425.267,Z 302.509,A -85,B 0,C 180,E1 -9663.048,E2 -9663.048} C_VEL
LIN {X 0,Y 425.276,Z 302.507,A -85,B 0,C 180,E1 -9665.927,E2 -9665.927} C_VEL
LIN {X 0,Y 425.256,Z 302.512,A -85,B 0,C 180,E1 -9669.036,E2 -9669.036} C_VEL
LIN {X 0,Y 425.251,Z 302.515,A -85,B 0,C 180,E1 -9672.655,E2 -9672.655} C_VEL
LIN {X 0,Y 425.28,Z 302.509,A -85,B 0,C 180,E1 -9675.282,E2 -9675.282} C_VEL
LIN {X 0,Y 425.242,Z 302.513,A -85,B 0,C 180,E1 -9678.617,E2 -9678.617} C_VEL
LIN {X 0,Y 425.272,Z 302.515,A -85,B 0,C 180,E1 -9681.098,E2 -9681.098} C_VEL
LIN {X 0,Y 425.285,Z 302.506,A -85,B 0,C 180,E1 -9684.662,E2 -9684.662} C_VEL
LIN {X 0,Y 425.238,Z 302.511,A -85,B 0,C 180,E1 -9688.07,E2 -9688.07} C_VEL
LIN {X 0,Y 425.284,Z 302.512,A -85,B 0,C 180,E1 -9691.364,E2 -9691.364} C_VEL
LIN {X 0,Y 425.243,Z 302.51,A -85,B 0,C 180,E1 -9694.551,E2 -9694.551} C_VEL
LIN {X 0,Y 425.284,Z 302.512,A -85,B 0,C 180,E1 -9697.729,E2 -9697.729} C_VEL
LIN {X 0,Y 425.35,Z 302.497,A -85,B 0,C 180,E1 -9700.703,E2 -9700.703} C_VEL
LIN {X 0,Y 425.3,Z 302.509,A -85,B 0,C 180,E1 -9703.684,E2 -9703.684} C_VEL
LIN {X 0,Y 425.392,Z 302.495,A -85,B 0,C 180,E1 -9707.597,E2 -9707.597} C_VEL
LIN {X 0,Y 425.385,Z 302.493,A -85,B 0,C 180,E1 -9711.449,E2 -9711.449} C_VEL
LIN {X 0,Y 425.498,Z 302.484,A -85,B 0,C 180,E1 -9714.312,E2 -9714.312} C_VEL
LIN {X 0,Y 425.558,Z 302.477,A -85,B 0,C 180,E1 -9718.107,E2 -9718.107} C_VEL
LIN {X 0,Y 425.499,Z 302.479,A -85,B 0,C 180,E1 -9720.946,E2 -9720.946} C_VEL
LIN {X 0,Y 425.508,Z 302.48,A -85,B 0,C 180,E1 -9722.84,E2 -9722.84} C_VEL
LIN {X 0,Y 425.531,Z 302.474,A -85,B 0,C 180,E1 -9725.687,E2 -9725.687} C_VEL
LIN {X 0,Y 425.397,Z 302.498,A -85,B 0,C 180,E1 -9728.551,E2 -9728.551} C_VEL
LIN {X 0,Y 425.402,Z 302.494,A -85,B 0,C 180,E1 -9732.402,E2 -9732.402} C_VEL
LIN {X 0,Y 425.379,Z 302.495,A -85,B 0,C 180,E1 -9736.312,E2 -9736.312} C_VEL
LIN {X 0,Y 425.319,Z 302.501,A -85,B 0,C 180,E1 -9739.636,E2 -9739.636} C_VEL
LIN {X 0,Y 425.279,Z 302.506,A -85,B 0,C 180,E1 -9742.339,E2 -9742.339} C_VEL
LIN {X 0,Y 425.31,Z 302.504,A -85,B 0,C 180,E1 -9744.657,E2 -9744.657} C_VEL
LIN {X 0,Y 425.337,Z 302.502,A -85,B 0,C 180,E1 -9747.558,E2 -9747.558} C_VEL
LIN {X 0,Y 425.28,Z 302.507,A -85,B 0,C 180,E1 -9750.817,E2 -9750.817} C_VEL
LIN {X 0,Y 425.304,Z 302.502,A -85,B 0,C 180,E1 -9754.288,E2 -9754.288} C_VEL
LIN {X 0,Y 425.269,Z 302.513,A -85,B 0,C 180,E1 -9757.695,E2 -9757.695} C_VEL
LIN {X 0,Y 425.259,Z 302.508,A -85,B 0,C 180,E1 -9760.519,E2 -9760.519} C_VEL
LIN {X 0,Y 425.25,Z 302.512,A -85,B 0,C 180,E1 -9763.351,E2 -9763.351} C_VEL
LIN {X 0,Y 425.255,Z 302.513,A -85,B 0,C 180,E1 -9766.045,E2 -9766.045} C_VEL
LIN {X 0,Y 425.271,Z 302.509,A -85,B 0,C 180,E1 -9769.481,E2 -9769.481} C_VEL
LIN {X 0,Y 425.272,Z 302.509,A -85,B 0,C 180,E1 -9772.49,E2 -9772.49} C_VEL
LIN {X 0,Y 425.304,Z 302.507,A -85,B 0,C 180,E1 -9775.818,E2 -9775.818} C_VEL
LIN {X 0,Y 425.288,Z 302.504,A -85,B 0,C 180,E1 -9779.24,E2 -9779.24} C_VEL
LIN {X 0,Y 425.343,Z 302.505,A -85,B 0,C 180,E1 -9782.443,E2 -9782.443} C_VEL
LIN {X 0,Y 425.366,Z 302.644,A -85,B 0,C 180,E1 -9783.412,E2 -9783.412} C_VEL
LIN {X 0,Y 427.841,Z 316.265,A -85,B 0,C 180,E1 -9786.269,E2 -9786.269} C_VEL
LIN {X 0,Y 427.024,Z 331.71,A -85,B 0,C 180,E1 -9789.278,E2 -9789.278} C_VEL
LIN {X 0,Y 426.4,Z 343.369,A -85,B 0,C 180,E1 -9791.526,E2 -9791.526} C_VEL
LIN {X 0,Y 430.021,Z 367.835,A -85,B 0,C 180,E1 -9792.087,E2 -9792.087} C_VEL
LIN {X 0,Y 429.192,Z 451.476,A -85,B 0,C 180,E1 -9793.502,E2 -9793.502} C_VEL
LIN {X 0,Y 428.67,Z 464.812,A -85,B 0,C 180,E1 -9793.909,E2 -9793.909} C_VEL
LIN {X 0,Y 428.227,Z 477.05,A -85,B 0,C 180,E1 -9794.472,E2 -9794.472} C_VEL
LIN {X 0,Y 427.543,Z 489.365,A -85,B 0,C 180,E1 -9795.24,E2 -9795.24} C_VEL
LIN {X 0,Y 426.817,Z 500.889,A -85,B 0,C 180,E1 -9796.177,E2 -9796.177} C_VEL
LIN {X 0,Y 426.179,Z 511.479,A -85,B 0,C 180,E1 -9797.259,E2 -9797.259} C_VEL
LIN {X 0,Y 425.652,Z 520.036,A -85,B 0,C 180,E1 -9798.332,E2 -9798.332} C_VEL
LIN {X 0,Y 425.064,Z 529.292,A -85,B 0,C 180,E1 -9799.763,E2 -9799.763} C_VEL
LIN {X 0,Y 424.682,Z 536.729,A -85,B 0,C 180,E1 -9801.196,E2 -9801.196} C_VEL
LIN {X 0,Y 424.349,Z 543.558,A -85,B 0,C 180,E1 -9802.865,E2 -9802.865} C_VEL
LIN {X 0,Y 424.189,Z 548.055,A -85,B 0,C 180,E1 -9804.296,E2 -9804.296} C_VEL
LIN {X 0,Y 424.199,Z 550.427,A -85,B 0,C 180,E1 -9805.249,E2 -9805.249} C_VEL
LIN {X 0,Y 424.099,Z 552.362,A -85,B 0,C 180,E1 -9806.2,E2 -9806.2} C_VEL
LIN {X 0,Y 424.132,Z 553.873,A -85,B 0,C 180,E1 -9807.151,E2 -9807.151} C_VEL
LIN {X 0,Y 424.128,Z 554.93,A -85,B 0,C 180,E1 -9808.102,E2 -9808.102} C_VEL
LIN {X 0,Y 424.084,Z 555.87,A -85,B 0,C 180,E1 -9810.001,E2 -9810.001} C_VEL
LIN {X 0,Y 424.088,Z 555.754,A -85,B 0,C 180,E1 -9810.95,E2 -9810.95} C_VEL
LIN {X 0,Y 424.128,Z 555.207,A -85,B 0,C 180,E1 -9811.9,E2 -9811.9} C_VEL
LIN {X 0,Y 424.13,Z 554.266,A -85,B 0,C 180,E1 -9812.85,E2 -9812.85} C_VEL
LIN {X 0,Y 424.098,Z 552.932,A -85,B 0,C 180,E1 -9813.801,E2 -9813.801} C_VEL
LIN {X 0,Y 424.207,Z 550.117,A -85,B 0,C 180,E1 -9815.229,E2 -9815.229} C_VEL
LIN {X 0,Y 424.301,Z 546.283,A -85,B 0,C 180,E1 -9816.659,E2 -9816.659} C_VEL
LIN {X 0,Y 424.548,Z 541.337,A -85,B 0,C 180,E1 -9818.09,E2 -9818.09} C_VEL
LIN {X 0,Y 424.951,Z 535.129,A -85,B 0,C 180,E1 -9819.52,E2 -9819.52} C_VEL
LIN {X 0,Y 425.45,Z 527.404,A -85,B 0,C 180,E1 -9820.952,E2 -9820.952} C_VEL
LIN {X 0,Y 426.288,Z 517.739,A -85,B 0,C 180,E1 -9822.376,E2 -9822.376} C_VEL
LIN {X 0,Y 426.996,Z 508.437,A -85,B 0,C 180,E1 -9823.491,E2 -9823.491} C_VEL
LIN {X 0,Y 427.625,Z 497.968,A -85,B 0,C 180,E1 -9824.516,E2 -9824.516} C_VEL
LIN {X 0,Y 428.518,Z 485.565,A -85,B 0,C 180,E1 -9825.457,E2 -9825.457} C_VEL
LIN {X 0,Y 429.26,Z 473.408,A -85,B 0,C 180,E1 -9826.161,E2 -9826.161} C_VEL
LIN {X 0,Y 429.842,Z 461.597,A -85,B 0,C 180,E1 -9826.657,E2 -9826.657} C_VEL
LIN {X 0,Y 430.201,Z 448.816,A -85,B 0,C 180,E1 -9827.01,E2 -9827.01} C_VEL
LIN {X 0,Y 431.132,Z 367.428,A -85,B 0,C 180,E1 -9828.397,E2 -9828.397} C_VEL
LIN {X 0,Y 426.952,Z 343.061,A -85,B 0,C 180,E1 -9829.055,E2 -9829.055} C_VEL
LIN {X 0,Y 428.093,Z 324.588,A -85,B 0,C 180,E1 -9832.694,E2 -9832.694} C_VEL
LIN {X 0,Y 428.442,Z 318.299,A -85,B 0,C 180,E1 -9833.953,E2 -9833.953} C_VEL
LIN {X 0,Y 426.599,Z 308.258,A -85,B 0,C 180,E1 -9836.149,E2 -9836.149} C_VEL
LIN {X 0,Y 425.381,Z 302.504,A -85,B 0,C 180,E1 -9837.464,E2 -9837.464} C_VEL
LIN {X 0,Y 425.29,Z 302.515,A -85,B 0,C 180,E1 -9840.816,E2 -9840.816} C_VEL
LIN {X 0,Y 425.313,Z 302.51,A -85,B 0,C 180,E1 -9844.288,E2 -9844.288} C_VEL
LIN {X 0,Y 425.278,Z 302.512,A -85,B 0,C 180,E1 -9847.695,E2 -9847.695} C_VEL
LIN {X 0,Y 425.267,Z 302.512,A -85,B 0,C 180,E1 -9850.518,E2 -9850.518} C_VEL
LIN {X 0,Y 425.257,Z 302.51,A -85,B 0,C 180,E1 -9853.351,E2 -9853.351} C_VEL
LIN {X 0,Y 425.262,Z 302.513,A -85,B 0,C 180,E1 -9856.044,E2 -9856.044} C_VEL
LIN {X 0,Y 425.266,Z 302.512,A -85,B 0,C 180,E1 -9858.62,E2 -9858.62} C_VEL
LIN {X 0,Y 425.282,Z 302.505,A -85,B 0,C 180,E1 -9861.1,E2 -9861.1} C_VEL
LIN {X 0,Y 425.3,Z 302.507,A -85,B 0,C 180,E1 -9864.664,E2 -9864.664} C_VEL
LIN {X 0,Y 425.265,Z 302.505,A -85,B 0,C 180,E1 -9868.073,E2 -9868.073} C_VEL
LIN {X 0,Y 425.315,Z 302.503,A -85,B 0,C 180,E1 -9871.367,E2 -9871.367} C_VEL
LIN {X 0,Y 425.271,Z 302.509,A -85,B 0,C 180,E1 -9874.553,E2 -9874.553} C_VEL
LIN {X 0,Y 425.284,Z 302.506,A -85,B 0,C 180,E1 -9876.634,E2 -9876.634} C_VEL
LIN {X 0,Y 425.296,Z 302.506,A -85,B 0,C 180,E1 -9879.695,E2 -9879.695} C_VEL
LIN {X 0,Y 425.334,Z 302.498,A -85,B 0,C 180,E1 -9882.697,E2 -9882.697} C_VEL
LIN {X 0,Y 425.348,Z 302.501,A -85,B 0,C 180,E1 -9885.65,E2 -9885.65} C_VEL
LIN {X 0,Y 425.35,Z 302.494,A -85,B 0,C 180,E1 -9888.564,E2 -9888.564} C_VEL
LIN {X 0,Y 425.507,Z 302.476,A -85,B 0,C 180,E1 -9892.311,E2 -9892.311} C_VEL
LIN {X 0,Y 425.547,Z 302.472,A -85,B 0,C 180,E1 -9894.313,E2 -9894.313} C_VEL
LIN {X 0,Y 425.57,Z 302.474,A -85,B 0,C 180,E1 -9898.107,E2 -9898.107} C_VEL
LIN {X 0,Y 425.698,Z 302.454,A -85,B 0,C 180,E1 -9900,E2 -9900} C_VEL
LIN {X 0,Y 425.537,Z 302.473,A -85,B 0,C 180,E1 -9902.84,E2 -9902.84} C_VEL
LIN {X 0,Y 425.498,Z 302.481,A -85,B 0,C 180,E1 -9906.524,E2 -9906.524} C_VEL
LIN {X 0,Y 425.4,Z 302.486,A -85,B 0,C 180,E1 -9909.51,E2 -9909.51} C_VEL
LIN {X 0,Y 425.395,Z 302.491,A -85,B 0,C 180,E1 -9912.904,E2 -9912.904} C_VEL
LIN {X 0,Y 425.363,Z 302.501,A -85,B 0,C 180,E1 -9916.605,E2 -9916.605} C_VEL
LIN {X 0,Y 425.33,Z 302.5,A -85,B 0,C 180,E1 -9919.636,E2 -9919.636} C_VEL
LIN {X 0,Y 425.29,Z 302.502,A -85,B 0,C 180,E1 -9922.339,E2 -9922.339} C_VEL
LIN {X 0,Y 425.322,Z 302.503,A -85,B 0,C 180,E1 -9924.657,E2 -9924.657} C_VEL
LIN {X 0,Y 425.302,Z 302.503,A -85,B 0,C 180,E1 -9927.561,E2 -9927.561} C_VEL
LIN {X 0,Y 425.29,Z 302.507,A -85,B 0,C 180,E1 -9930.816,E2 -9930.816} C_VEL
LIN {X 0,Y 425.312,Z 302.5,A -85,B 0,C 180,E1 -9934.288,E2 -9934.288} C_VEL
LIN {X 0,Y 425.279,Z 302.511,A -85,B 0,C 180,E1 -9937.695,E2 -9937.695} C_VEL
LIN {X 0,Y 425.279,Z 302.508,A -85,B 0,C 180,E1 -9940.52,E2 -9940.52} C_VEL
LIN {X 0,Y 425.264,Z 302.513,A -85,B 0,C 180,E1 -9943.956,E2 -9943.956} C_VEL
LIN {X 0,Y 425.253,Z 302.513,A -85,B 0,C 180,E1 -9946.65,E2 -9946.65} C_VEL
LIN {X 0,Y 425.247,Z 302.513,A -85,B 0,C 180,E1 -9949.868,E2 -9949.868} C_VEL
LIN {X 0,Y 425.279,Z 302.511,A -85,B 0,C 180,E1 -9952.489,E2 -9952.489} C_VEL
LIN {X 0,Y 425.347,Z 302.618,A -85,B 0,C 180,E1 -9955.856,E2 -9955.856} C_VEL
LIN {X 0,Y 427.367,Z 312.898,A -85,B 0,C 180,E1 -9958.248,E2 -9958.248} C_VEL
LIN {X 0,Y 427.179,Z 321.036,A -85,B 0,C 180,E1 -9959.991,E2 -9959.991} C_VEL
LIN {X 0,Y 431.295,Z 340.094,A -85,B 0,C 180,E1 -9960.563,E2 -9960.563} C_VEL
LIN {X 0,Y 431.259,Z 355.589,A -85,B 0,C 180,E1 -9960.833,E2 -9960.833} C_VEL
LIN {X 0,Y 430.312,Z 429.095,A -85,B 0,C 180,E1 -9962.1,E2 -9962.1} C_VEL
LIN {X 0,Y 429.938,Z 440.829,A -85,B 0,C 180,E1 -9962.462,E2 -9962.462} C_VEL
LIN {X 0,Y 429.351,Z 453.686,A -85,B 0,C 180,E1 -9963.049,E2 -9963.049} C_VEL
LIN {X 0,Y 428.828,Z 464.733,A -85,B 0,C 180,E1 -9963.736,E2 -9963.736} C_VEL
LIN {X 0,Y 428.072,Z 476.439,A -85,B 0,C 180,E1 -9964.673,E2 -9964.673} C_VEL
LIN {X 0,Y 427.274,Z 486.805,A -85,B 0,C 180,E1 -9965.719,E2 -9965.719} C_VEL
LIN {X 0,Y 426.531,Z 496.447,A -85,B 0,C 180,E1 -9966.921,E2 -9966.921} C_VEL
LIN {X 0,Y 425.886,Z 504.791,A -85,B 0,C 180,E1 -9968.204,E2 -9968.204} C_VEL
LIN {X 0,Y 425.321,Z 512.578,A -85,B 0,C 180,E1 -9969.695,E2 -9969.695} C_VEL
LIN {X 0,Y 424.836,Z 518.772,A -85,B 0,C 180,E1 -9971.18,E2 -9971.18} C_VEL
LIN {X 0,Y 424.508,Z 523.623,A -85,B 0,C 180,E1 -9972.662,E2 -9972.662} C_VEL
LIN {X 0,Y 424.367,Z 526.655,A -85,B 0,C 180,E1 -9973.854,E2 -9973.854} C_VEL
LIN {X 0,Y 424.105,Z 529.88,A -85,B 0,C 180,E1 -9975.607,E2 -9975.607} C_VEL
LIN {X 0,Y 424.066,Z 531.015,A -85,B 0,C 180,E1 -9976.534,E2 -9976.534} C_VEL
LIN {X 0,Y 423.396,Z 531.806,A -85,B 0,C 180,E1 -9977.321,E2 -9977.321} C_VEL
LIN {X 0,Y 420.479,Z 532.381,A -85,B 0,C 180,E1 -9978.607,E2 -9978.607} C_VEL
LIN {X 0,Y 418.019,Z 532.222,A -85,B 0,C 180,E1 -9979.648,E2 -9979.648} C_VEL
LIN {X 0,Y 416.924,Z 531.698,A -85,B 0,C 180,E1 -9980.587,E2 -9980.587} C_VEL
LIN {X 0,Y 416.907,Z 531.552,A -85,B 0,C 180,E1 -9980.723,E2 -9980.723} C_VEL
LIN {X 0,Y 417.039,Z 529.838,A -85,B 0,C 180,E1 -9982.251,E2 -9982.251} C_VEL
LIN {X 0,Y 417.199,Z 527.286,A -85,B 0,C 180,E1 -9983.671,E2 -9983.671} C_VEL
LIN {X 0,Y 417.311,Z 523.547,A -85,B 0,C 180,E1 -9985.169,E2 -9985.169} C_VEL
LIN {X 0,Y 417.576,Z 518.787,A -85,B 0,C 180,E1 -9986.622,E2 -9986.622} C_VEL
LIN {X 0,Y 417.821,Z 512.796,A -85,B 0,C 180,E1 -9988.071,E2 -9988.071} C_VEL
LIN {X 0,Y 418.444,Z 505.319,A -85,B 0,C 180,E1 -9989.518,E2 -9989.518} C_VEL
LIN {X 0,Y 418.887,Z 497.723,A -85,B 0,C 180,E1 -9990.72,E2 -9990.72} C_VEL
LIN {X 0,Y 419.4,Z 488.517,A -85,B 0,C 180,E1 -9991.92,E2 -9991.92} C_VEL
LIN {X 0,Y 420.191,Z 478.228,A -85,B 0,C 180,E1 -9992.995,E2 -9992.995} C_VEL
LIN {X 0,Y 420.899,Z 466.847,A -85,B 0,C 180,E1 -9993.949,E2 -9993.949} C_VEL
LIN {X 0,Y 421.437,Z 455.007,A -85,B 0,C 180,E1 -9994.722,E2 -9994.722} C_VEL
LIN {X 0,Y 421.885,Z 441.878,A -85,B 0,C 180,E1 -9995.346,E2 -9995.346} C_VEL
LIN {X 0,Y 422.238,Z 428.794,A -85,B 0,C 180,E1 -9995.761,E2 -9995.761} C_VEL
LIN {X 0,Y 423.323,Z 341.628,A -85,B 0,C 180,E1 -9997.257,E2 -9997.257} C_VEL
LIN {X 0,Y 419.663,Z 321.305,A -85,B 0,C 180,E1 -9997.759,E2 -9997.759} C_VEL
LIN {X 0,Y 420.002,Z 312.658,A -85,B 0,C 180,E1 -9999.632,E2 -9999.632} C_VEL
LIN {X 0,Y 418.388,Z 303.371,A -85,B 0,C 180,E1 -10001.812,E2 -10001.812} C_VEL
LIN {X 0,Y 418.281,Z 303.38,A -85,B 0,C 180,E1 -10004.597,E2 -10004.597} C_VEL
LIN {X 0,Y 418.258,Z 303.383,A -85,B 0,C 180,E1 -10007.604,E2 -10007.604} C_VEL
LIN {X 0,Y 418.251,Z 303.383,A -85,B 0,C 180,E1 -10010.662,E2 -10010.662} C_VEL
LIN {X 0,Y 418.257,Z 303.383,A -85,B 0,C 180,E1 -10013.782,E2 -10013.782} C_VEL
LIN {X 0,Y 418.206,Z 303.387,A -85,B 0,C 180,E1 -10017.041,E2 -10017.041} C_VEL
LIN {X 0,Y 418.237,Z 303.389,A -85,B 0,C 180,E1 -10020.272,E2 -10020.272} C_VEL
LIN {X 0,Y 418.231,Z 303.384,A -85,B 0,C 180,E1 -10023.678,E2 -10023.678} C_VEL
LIN {X 0,Y 418.232,Z 303.385,A -85,B 0,C 180,E1 -10027.224,E2 -10027.224} C_VEL
LIN {X 0,Y 418.203,Z 303.394,A -85,B 0,C 180,E1 -10030.866,E2 -10030.866} C_VEL
LIN {X 0,Y 418.197,Z 303.388,A -85,B 0,C 180,E1 -10033.727,E2 -10033.727} C_VEL
LIN {X 0,Y 418.193,Z 303.39,A -85,B 0,C 180,E1 -10036.446,E2 -10036.446} C_VEL
LIN {X 0,Y 418.201,Z 303.394,A -85,B 0,C 180,E1 -10039.132,E2 -10039.132} C_VEL
LIN {X 0,Y 418.227,Z 303.387,A -85,B 0,C 180,E1 -10042.774,E2 -10042.774} C_VEL
LIN {X 0,Y 418.221,Z 303.385,A -85,B 0,C 180,E1 -10046.32,E2 -10046.32} C_VEL
LIN {X 0,Y 418.226,Z 303.387,A -85,B 0,C 180,E1 -10049.726,E2 -10049.726} C_VEL
LIN {X 0,Y 418.192,Z 303.391,A -85,B 0,C 180,E1 -10053.015,E2 -10053.015} C_VEL
LIN {X 0,Y 418.247,Z 303.383,A -85,B 0,C 180,E1 -10056.216,E2 -10056.216} C_VEL
LIN {X 0,Y 418.24,Z 303.386,A -85,B 0,C 180,E1 -10059.336,E2 -10059.336} C_VEL
LIN {X 0,Y 418.232,Z 303.384,A -85,B 0,C 180,E1 -10062.393,E2 -10062.393} C_VEL
